C05472=1136.508,344.790,-80.424,-177.368,10.885,149.505
C05473=1136.503,345.037,-80.459,-177.365,10.887,149.505
C05474=1136.500,345.285,-80.494,-177.361,10.890,149.505
C05475=1136.495,345.532,-80.529,-177.358,10.892,149.504
C05476=1136.492,345.780,-80.563,-177.355,10.895,149.504
C05477=1136.488,346.027,-80.598,-177.351,10.897,149.504
C05478=1136.484,346.275,-80.633,-177.348,10.899,149.504
C05479=1136.480,346.523,-80.668,-177.345,10.902,149.503
C05480=1136.476,346.770,-80.702,-177.342,10.905,149.503
C05481=1136.472,347.018,-80.737,-177.338,10.907,149.503
C05482=1136.468,347.265,-80.772,-177.335,10.910,149.503
C05483=1136.464,347.513,-80.807,-177.332,10.912,149.503
C05484=1136.460,347.761,-80.842,-177.328,10.915,149.503
C05485=1136.458,347.974,-80.872,-177.325,10.917,149.502
C05486=1136.454,348.186,-80.902,-177.323,10.919,149.502
C05487=1136.450,348.400,-80.932,-177.320,10.921,149.502
C05488=1136.447,348.614,-80.963,-177.317,10.923,149.502
C05489=1136.443,348.827,-80.993,-177.314,10.926,149.502
C05490=1136.440,349.040,-81.022,-177.311,10.928,149.501
C05491=1136.437,349.254,-81.053,-177.309,10.930,149.501
C05492=1136.433,349.466,-81.083,-177.306,10.932,149.501
C05493=1136.429,349.714,-81.118,-177.302,10.935,149.501
C05494=1136.425,349.962,-81.154,-177.298,10.937,149.501
C05495=1136.421,350.209,-81.189,-177.294,10.941,149.500
C05496=1136.417,350.457,-81.224,-177.291,10.943,149.500
C05497=1136.413,350.704,-81.259,-177.286,10.946,149.500
C05498=1136.410,350.951,-81.293,-177.283,10.949,149.499
C05499=1136.406,351.199,-81.329,-177.279,10.952,149.499
C05500=1136.402,351.446,-81.364,-177.275,10.954,149.499
C05501=1136.399,351.694,-81.400,-177.272,10.957,149.499
C05502=1136.394,351.941,-81.434,-177.268,10.960,149.498
C05503=1136.390,352.189,-81.470,-177.264,10.962,149.498
C05504=1136.387,352.436,-81.505,-177.261,10.965,149.498
C05505=1136.383,352.684,-81.541,-177.257,10.967,149.498
C05506=1136.378,352.931,-81.575,-177.253,10.970,149.497
C05507=1136.375,353.179,-81.611,-177.250,10.973,149.497
C05508=1136.371,353.426,-81.646,-177.245,10.976,149.497
C05509=1136.368,353.674,-81.682,-177.242,10.978,149.496
C05510=1136.363,353.921,-81.717,-177.239,10.981,149.496
C05511=1136.359,354.169,-81.752,-177.234,10.984,149.496
C05512=1136.355,354.416,-81.788,-177.231,10.986,149.496
C05513=1136.351,354.664,-81.824,-177.228,10.988,149.495
C05514=1136.347,354.911,-81.859,-177.223,10.991,149.495
C05515=1136.343,355.158,-81.894,-177.220,10.994,149.495
C05516=1136.340,355.406,-81.930,-177.217,10.996,149.495
C05517=1136.336,355.653,-81.965,-177.213,10.998,149.494
C05518=1136.332,355.901,-82.001,-177.209,11.002,149.494
C05519=1136.329,356.148,-82.036,-177.206,11.004,149.494
C05520=1136.324,356.395,-82.072,-177.202,11.006,149.493
C05521=1136.320,356.643,-82.108,-177.199,11.009,149.493
C05522=1136.316,356.890,-82.143,-177.195,11.012,149.493
C05523=1136.313,357.138,-82.179,-177.191,11.014,149.493
C05524=1136.309,357.385,-82.214,-177.188,11.017,149.492
C05525=1136.305,357.633,-82.250,-177.184,11.019,149.492
C05526=1136.301,357.881,-82.286,-177.181,11.022,149.492
C05527=1136.297,358.127,-82.321,-177.177,11.024,149.492
C05528=1136.293,358.374,-82.358,-177.174,11.027,149.491
C05529=1136.290,358.622,-82.393,-177.170,11.029,149.491
C05530=1136.285,358.870,-82.429,-177.167,11.032,149.491
C05531=1136.282,359.117,-82.465,-177.163,11.034,149.490
C05532=1136.278,359.365,-82.500,-177.160,11.036,149.490
C05533=1136.275,359.612,-82.537,-177.157,11.039,149.490
C05534=1136.270,359.859,-82.573,-177.153,11.041,149.490
C05535=1136.266,360.107,-82.608,-177.150,11.044,149.489
C05536=1136.263,360.354,-82.644,-177.146,11.046,149.489
C05537=1136.259,360.601,-82.680,-177.143,11.048,149.489
C05538=1136.254,360.848,-82.716,-177.139,11.051,149.489
C05539=1136.251,361.096,-82.751,-177.135,11.054,149.488
C05540=1136.247,361.343,-82.787,-177.132,11.056,149.488
C05541=1136.243,361.556,-82.819,-177.129,11.058,149.488
C05542=1136.241,361.770,-82.850,-177.127,11.060,149.488
C05543=1136.238,361.983,-82.881,-177.123,11.062,149.487
C05544=1136.234,362.196,-82.912,-177.121,11.064,149.487
C05545=1136.231,362.409,-82.943,-177.117,11.066,149.487
C05546=1136.228,362.622,-82.973,-177.115,11.068,149.487
C05547=1136.224,362.835,-83.005,-177.111,11.070,149.486
C05548=1136.221,363.048,-83.036,-177.109,11.072,149.486
C05549=1136.217,363.295,-83.072,-177.105,11.075,149.486
C05550=1136.213,363.543,-83.108,-177.102,11.077,149.486
C05551=1136.210,363.790,-83.145,-177.099,11.080,149.486
C05552=1136.205,364.038,-83.181,-177.096,11.082,149.485
C05553=1136.202,364.285,-83.217,-177.092,11.085,149.485
C05554=1136.198,364.532,-83.253,-177.090,11.086,149.485
C05555=1136.194,364.779,-83.289,-177.086,11.088,149.484
C05556=1136.190,365.027,-83.325,-177.083,11.091,149.484
C05557=1136.186,365.274,-83.362,-177.079,11.093,149.484
C05558=1136.183,365.522,-83.397,-177.076,11.096,149.484
C05559=1136.179,365.769,-83.434,-177.073,11.098,149.484
C05560=1136.175,366.016,-83.470,-177.069,11.101,149.483
C05561=1136.171,366.263,-83.507,-177.067,11.102,149.483
C05562=1136.168,366.511,-83.543,-177.063,11.105,149.483
C05563=1136.164,366.759,-83.579,-177.060,11.107,149.483
C05564=1136.160,367.006,-83.616,-177.057,11.110,149.483
C05565=1136.156,367.253,-83.653,-177.053,11.112,149.482
C05566=1136.153,367.500,-83.688,-177.051,11.114,149.482
C05567=1136.148,367.748,-83.725,-177.047,11.116,149.482
C05568=1136.144,367.995,-83.762,-177.044,11.119,149.482
C05569=1136.141,368.242,-83.797,-177.041,11.121,149.481
C05570=1136.137,368.490,-83.834,-177.038,11.123,149.481
C05571=1136.133,368.736,-83.870,-177.035,11.126,149.481
C05572=1136.129,368.984,-83.907,-177.032,11.128,149.481
C05573=1136.125,369.232,-83.944,-177.029,11.130,149.481
C05574=1136.122,369.479,-83.980,-177.026,11.132,149.480
C05575=1136.118,369.726,-84.017,-177.022,11.135,149.480
C05576=1136.115,369.973,-84.053,-177.020,11.136,149.480
C05577=1136.110,370.220,-84.090,-177.016,11.139,149.480
C05578=1136.106,370.468,-84.126,-177.013,11.141,149.479
C05579=1136.103,370.715,-84.162,-177.010,11.143,149.479
C05580=1136.099,370.962,-84.199,-177.007,11.146,149.479
C05581=1136.095,371.210,-84.237,-177.004,11.148,149.479
C05582=1136.092,371.457,-84.273,-177.001,11.150,149.479
C05583=1136.088,371.704,-84.310,-176.998,11.152,149.479
C05584=1136.084,371.951,-84.347,-176.995,11.155,149.478
C05585=1136.079,372.198,-84.383,-176.992,11.157,149.478
C05586=1136.076,372.445,-84.420,-176.989,11.159,149.478
C05587=1136.073,372.693,-84.457,-176.987,11.161,149.478
C05588=1136.068,372.940,-84.494,-176.983,11.164,149.478
C05589=1136.065,373.187,-84.530,-176.980,11.166,149.477
C05590=1136.061,373.434,-84.567,-176.978,11.168,149.477
C05591=1136.057,373.682,-84.604,-176.974,11.171,149.477
C05592=1136.053,373.930,-84.641,-176.972,11.172,149.477
C05593=1136.049,374.177,-84.678,-176.969,11.175,149.477
C05594=1136.046,374.424,-84.714,-176.966,11.177,149.477
C05595=1136.042,374.671,-84.751,-176.963,11.179,149.476
C05596=1136.038,374.919,-84.788,-176.961,11.181,149.476
C05597=1136.035,375.131,-84.819,-176.958,11.183,149.476
C05598=1136.032,375.344,-84.851,-176.956,11.185,149.476
C05599=1136.028,375.557,-84.883,-176.953,11.187,149.476
C05600=1136.025,375.771,-84.915,-176.951,11.189,149.476
C05601=1136.022,375.983,-84.947,-176.948,11.191,149.476
C05602=1136.019,376.196,-84.979,-176.946,11.193,149.476
C05603=1136.016,376.409,-85.011,-176.944,11.195,149.475
C05604=1136.012,376.622,-85.043,-176.941,11.197,149.475
C05605=1136.008,376.869,-85.079,-176.938,11.199,149.475
C05606=1136.004,377.116,-85.116,-176.936,11.201,149.475
C05607=1136.001,377.364,-85.154,-176.933,11.204,149.475
C05608=1135.997,377.611,-85.191,-176.930,11.206,149.475
C05609=1135.993,377.858,-85.228,-176.927,11.208,149.475
C05610=1135.990,378.106,-85.265,-176.925,11.210,149.475
C05611=1135.986,378.353,-85.302,-176.922,11.212,149.474
C05612=1135.982,378.600,-85.339,-176.919,11.215,149.474
C05613=1135.978,378.847,-85.376,-176.917,11.217,149.474
C05614=1135.974,379.095,-85.413,-176.914,11.219,149.474
C05615=1135.971,379.341,-85.450,-176.912,11.221,149.474
C05616=1135.967,379.588,-85.487,-176.909,11.223,149.474
C05617=1135.963,379.836,-85.524,-176.906,11.226,149.474
C05618=1135.960,380.083,-85.562,-176.904,11.228,149.474
C05619=1135.956,380.330,-85.599,-176.901,11.230,149.474
C05620=1135.952,380.578,-85.636,-176.899,11.233,149.474
C05621=1135.948,380.824,-85.674,-176.896,11.235,149.473
C05622=1135.944,381.072,-85.710,-176.894,11.237,149.473
C05623=1135.941,381.319,-85.748,-176.891,11.239,149.473
C05624=1135.937,381.566,-85.785,-176.888,11.241,149.473
C05625=1135.933,381.813,-85.822,-176.886,11.243,149.473
C05626=1135.930,382.060,-85.860,-176.883,11.246,149.473
C05627=1135.925,382.308,-85.897,-176.881,11.248,149.473
C05628=1135.922,382.554,-85.934,-176.879,11.250,149.473
C05629=1135.918,382.802,-85.972,-176.876,11.253,149.473
C05630=1135.914,383.049,-86.009,-176.874,11.255,149.473
C05631=1135.911,383.297,-86.046,-176.871,11.257,149.473
C05632=1135.907,383.543,-86.084,-176.869,11.260,149.473
C05633=1135.902,383.791,-86.122,-176.869,11.260,149.473
C05634=1135.899,384.038,-86.159,-176.868,11.262,149.473
C05635=1135.895,384.285,-86.196,-176.867,11.264,149.474
C05636=1135.891,384.532,-86.234,-176.866,11.265,149.474
C05637=1135.888,384.780,-86.271,-176.865,11.266,149.474
C05638=1135.884,385.026,-86.309,-176.864,11.268,149.474
C05639=1135.881,385.273,-86.347,-176.863,11.269,149.474
C05640=1135.877,385.521,-86.383,-176.862,11.271,149.474
C05641=1135.873,385.767,-86.421,-176.862,11.273,149.475
C05642=1135.869,386.015,-86.458,-176.861,11.273,149.475
C05643=1135.866,386.262,-86.496,-176.860,11.275,149.475
C05644=1135.862,386.510,-86.533,-176.859,11.277,149.475
C05645=1135.858,386.756,-86.571,-176.858,11.279,149.475
C05646=1135.854,387.004,-86.609,-176.858,11.280,149.476
C05647=1135.850,387.251,-86.646,-176.857,11.282,149.476
C05648=1135.847,387.497,-86.684,-176.856,11.284,149.476
C05649=1135.843,387.745,-86.721,-176.856,11.285,149.476
C05650=1135.839,387.992,-86.758,-176.855,11.287,149.477
C05651=1135.836,388.239,-86.796,-176.854,11.289,149.477
C05652=1135.832,388.486,-86.833,-176.854,11.290,149.477
C05653=1135.828,388.699,-86.866,-176.853,11.292,149.478
C05654=1135.825,388.912,-86.898,-176.853,11.293,149.478
C05655=1135.822,389.125,-86.931,-176.852,11.295,149.478
C05656=1135.820,389.337,-86.963,-176.852,11.296,149.478
C05657=1135.816,389.550,-86.995,-176.852,11.297,149.478
C05658=1135.813,389.763,-87.028,-176.851,11.299,149.479
C05659=1135.809,389.976,-87.060,-176.851,11.300,149.479
C05660=1135.806,390.189,-87.092,-176.850,11.302,149.479
C05661=1135.803,390.436,-87.130,-176.850,11.304,149.480
C05662=1135.798,390.683,-87.167,-176.850,11.306,149.480
C05663=1135.795,390.931,-87.205,-176.849,11.308,149.480
C05664=1135.791,391.177,-87.243,-176.849,11.309,149.481
C05665=1135.788,391.425,-87.280,-176.849,11.311,149.481
C05666=1135.784,391.672,-87.317,-176.848,11.314,149.482
C05667=1135.780,391.919,-87.356,-176.848,11.315,149.482
C05668=1135.776,392.166,-87.393,-176.847,11.317,149.482
C05669=1135.773,392.414,-87.431,-176.847,11.319,149.483
C05670=1135.769,392.660,-87.468,-176.847,11.321,149.483
C05671=1135.765,392.907,-87.505,-176.847,11.323,149.484
C05672=1135.762,393.155,-87.543,-176.847,11.325,149.484
C05673=1135.757,393.402,-87.581,-176.847,11.327,149.485
C05674=1135.754,393.649,-87.619,-176.846,11.329,149.485
C05675=1135.750,393.896,-87.656,-176.846,11.331,149.486
C05676=1135.747,394.143,-87.694,-176.846,11.333,149.486
C05677=1135.743,394.390,-87.732,-176.846,11.335,149.487
C05678=1135.739,394.638,-87.769,-176.845,11.338,149.487
C05679=1135.735,394.885,-87.807,-176.846,11.339,149.488
C05680=1135.732,395.132,-87.845,-176.846,11.342,149.488
C05681=1135.728,395.378,-87.882,-176.845,11.344,149.489
C05682=1135.724,395.626,-87.919,-176.846,11.346,149.490
C05683=1135.720,395.873,-87.958,-176.846,11.348,149.490
C05684=1135.716,396.120,-87.995,-176.845,11.351,149.491
C05685=1135.713,396.367,-88.033,-176.845,11.353,149.491
C05686=1135.709,396.614,-88.070,-176.846,11.355,149.492
C05687=1135.706,396.862,-88.108,-176.846,11.358,149.493
C05688=1135.701,397.108,-88.146,-176.846,11.360,149.493
C05689=1135.698,397.356,-88.184,-176.846,11.362,149.494
C05690=1135.694,397.603,-88.221,-176.846,11.364,149.495
C05691=1135.691,397.850,-88.259,-176.846,11.367,149.495
C05692=1135.687,398.097,-88.297,-176.847,11.369,149.496
C05693=1135.683,398.344,-88.335,-176.847,11.371,149.496
C05694=1135.679,398.591,-88.373,-176.847,11.374,149.497
C05695=1135.676,398.839,-88.410,-176.847,11.377,149.498
C05696=1135.672,399.085,-88.448,-176.848,11.379,149.499
C05697=1135.668,399.333,-88.486,-176.848,11.381,149.499
C05698=1135.664,399.579,-88.524,-176.848,11.384,149.500
C05699=1135.661,399.827,-88.562,-176.848,11.387,149.501
C05700=1135.657,400.074,-88.598,-176.849,11.389,149.502
C05701=1135.653,400.321,-88.637,-176.849,11.392,149.502
C05702=1135.649,400.568,-88.675,-176.850,11.395,149.503
C05703=1135.646,400.815,-88.712,-176.851,11.397,149.504
C05704=1135.642,401.062,-88.750,-176.851,11.400,149.505
C05705=1135.638,401.309,-88.787,-176.851,11.403,149.506
C05706=1135.634,401.557,-88.825,-176.852,11.406,149.507
C05707=1135.631,401.803,-88.863,-176.853,11.408,149.507
C05708=1135.627,402.051,-88.901,-176.853,11.411,149.508
C05709=1135.624,402.263,-88.934,-176.853,11.413,149.509
C05710=1135.621,402.476,-88.967,-176.854,11.416,149.510
C05711=1135.617,402.689,-88.998,-176.854,11.418,149.510
C05712=1135.614,402.902,-89.031,-176.855,11.420,149.511
C05713=1135.611,403.114,-89.064,-176.855,11.423,149.512
C05714=1135.608,403.327,-89.097,-176.856,11.425,149.513
C05715=1135.605,403.540,-89.129,-176.857,11.428,149.514
C05716=1135.601,403.753,-89.162,-176.858,11.430,149.514
C05717=1135.598,404.000,-89.199,-176.858,11.433,149.515
C05718=1135.594,404.247,-89.237,-176.859,11.436,149.516
C05719=1135.591,404.494,-89.275,-176.859,11.439,149.517
C05720=1135.587,404.741,-89.313,-176.860,11.443,149.518
C05721=1135.583,404.988,-89.351,-176.861,11.445,149.519
C05722=1135.580,405.235,-89.389,-176.862,11.448,149.520
C05723=1135.576,405.482,-89.426,-176.863,11.452,149.521
C05724=1135.572,405.730,-89.464,-176.864,11.455,149.522
C05725=1135.568,405.977,-89.502,-176.865,11.458,149.523
C05726=1135.565,406.224,-89.540,-176.865,11.462,149.525
C05727=1135.560,406.471,-89.578,-176.867,11.464,149.525
C05728=1135.557,406.718,-89.616,-176.868,11.468,149.527
C05729=1135.553,406.965,-89.653,-176.868,11.471,149.528
C05730=1135.550,407.212,-89.691,-176.869,11.474,149.529
C05731=1135.546,407.459,-89.730,-176.871,11.478,149.530
C05732=1135.542,407.707,-89.767,-176.872,11.481,149.531
C05733=1135.538,407.953,-89.804,-176.872,11.485,149.532
C05734=1135.534,408.201,-89.843,-176.874,11.487,149.533
C05735=1135.531,408.447,-89.880,-176.875,11.491,149.535
C05736=1135.527,408.695,-89.918,-176.876,11.494,149.536
C05737=1135.524,408.942,-89.956,-176.877,11.498,149.537
C05738=1135.520,409.189,-89.995,-176.878,11.502,149.538
C05739=1135.516,409.436,-90.032,-176.880,11.505,149.540
C05740=1135.513,409.683,-90.070,-176.881,11.509,149.541
C05741=1135.509,409.930,-90.109,-176.882,11.513,149.542
C05742=1135.505,410.177,-90.146,-176.884,11.516,149.543
C05743=1135.502,410.424,-90.184,-176.885,11.520,149.545
C05744=1135.497,410.671,-90.222,-176.887,11.523,149.546
C05745=1135.494,410.919,-90.259,-176.888,11.527,149.547
C05746=1135.490,411.165,-90.297,-176.889,11.530,149.549
C05747=1135.487,411.413,-90.335,-176.891,11.534,149.550
C05748=1135.482,411.659,-90.373,-176.892,11.538,149.551
C05749=1135.479,411.907,-90.411,-176.894,11.542,149.553
C05750=1135.475,412.153,-90.449,-176.895,11.546,149.554
C05751=1135.471,412.401,-90.487,-176.897,11.550,149.555
C05752=1135.468,412.648,-90.525,-176.898,11.554,149.557
C05753=1135.464,412.895,-90.563,-176.900,11.558,149.558
C05754=1135.460,413.142,-90.601,-176.902,11.562,149.560
C05755=1135.457,413.389,-90.639,-176.903,11.566,149.561
C05756=1135.453,413.636,-90.677,-176.905,11.570,149.563
C05757=1135.449,413.883,-90.715,-176.907,11.574,149.564
C05758=1135.446,414.130,-90.753,-176.908,11.578,149.566
C05759=1135.442,414.377,-90.790,-176.910,11.582,149.567
C05760=1135.439,414.624,-90.828,-176.912,11.586,149.569
C05761=1135.437,414.872,-90.866,-176.914,11.591,149.570
C05762=1135.434,415.119,-90.903,-176.916,11.595,149.572
C05763=1135.434,415.365,-90.941,-176.918,11.599,149.573
C05764=1135.433,415.614,-90.979,-176.919,11.603,149.575
C05765=1135.433,415.826,-91.011,-176.921,11.607,149.576
C05766=1135.434,416.039,-91.044,-176.922,11.611,149.578
C05767=1135.435,416.251,-91.075,-176.925,11.615,149.579
C05768=1135.436,416.464,-91.107,-176.926,11.618,149.581
C05769=1135.439,416.677,-91.139,-176.928,11.622,149.582
C05770=1135.441,416.889,-91.171,-176.930,11.626,149.584
C05771=1135.444,417.102,-91.203,-176.932,11.630,149.585
C05772=1135.448,417.314,-91.234,-176.934,11.634,149.586
C05773=1135.029,417.314,-91.297,-176.926,11.638,149.586
C05774=1135.025,417.102,-91.266,-176.924,11.634,149.584
C05775=1135.022,416.889,-91.234,-176.922,11.631,149.583
C05776=1135.019,416.676,-91.202,-176.920,11.627,149.581
C05777=1135.018,416.463,-91.170,-176.919,11.623,149.580
C05778=1135.016,416.251,-91.138,-176.917,11.619,149.578
C05779=1135.015,416.038,-91.106,-176.915,11.616,149.577
C05780=1135.014,415.826,-91.074,-176.914,11.612,149.576
C05781=1135.014,415.614,-91.041,-176.912,11.608,149.574
C05782=1135.015,415.365,-91.004,-176.910,11.603,149.573
C05783=1135.016,415.119,-90.966,-176.908,11.599,149.571
C05784=1135.017,414.871,-90.928,-176.906,11.595,149.570
C05785=1135.020,414.624,-90.891,-176.905,11.591,149.568
C05786=1135.023,414.377,-90.852,-176.903,11.587,149.567
C05787=1135.026,414.130,-90.815,-176.901,11.583,149.565
C05788=1135.030,413.884,-90.777,-176.900,11.578,149.563
C05789=1135.034,413.636,-90.738,-176.899,11.574,149.562
C05790=1135.037,413.389,-90.701,-176.897,11.570,149.560
C05791=1135.041,413.142,-90.663,-176.895,11.566,149.559
C05792=1135.044,412.895,-90.624,-176.894,11.562,149.558
C05793=1135.048,412.648,-90.587,-176.892,11.558,149.556
C05794=1135.052,412.400,-90.550,-176.890,11.554,149.555
C05795=1135.056,412.153,-90.511,-176.889,11.550,149.553
C05796=1135.059,411.906,-90.473,-176.887,11.546,149.552
C05797=1135.063,411.659,-90.436,-176.886,11.542,149.551
C05798=1135.067,411.412,-90.397,-176.885,11.538,149.549
C05799=1135.071,411.165,-90.360,-176.883,11.535,149.548
C05800=1135.074,410.918,-90.322,-176.882,11.531,149.547
C05801=1135.079,410.671,-90.284,-176.880,11.527,149.545
C05802=1135.082,410.424,-90.246,-176.879,11.523,149.544
C05803=1135.085,410.177,-90.208,-176.878,11.519,149.543
C05804=1135.090,409.930,-90.170,-176.877,11.516,149.542
C05805=1135.093,409.682,-90.132,-176.876,11.512,149.540
C05806=1135.097,409.436,-90.094,-176.874,11.508,149.539
C05807=1135.101,409.188,-90.056,-176.873,11.505,149.538
C05808=1135.104,408.942,-90.018,-176.872,11.501,149.537
C05809=1135.107,408.694,-89.980,-176.871,11.498,149.535
C05810=1135.111,408.448,-89.942,-176.870,11.494,149.534
C05811=1135.115,408.200,-89.904,-176.869,11.491,149.533
C05812=1135.119,407.954,-89.866,-176.868,11.487,149.532
C05813=1135.122,407.706,-89.828,-176.867,11.484,149.531
C05814=1135.127,407.459,-89.791,-176.866,11.480,149.530
C05815=1135.130,407.212,-89.753,-176.864,11.478,149.528
C05816=1135.133,406.964,-89.715,-176.863,11.474,149.527
C05817=1135.138,406.718,-89.677,-176.862,11.471,149.526
C05818=1135.141,406.470,-89.639,-176.862,11.468,149.525
C05819=1135.145,406.224,-89.601,-176.861,11.464,149.524
C05820=1135.148,405.976,-89.563,-176.860,11.461,149.523
C05821=1135.153,405.730,-89.525,-176.859,11.458,149.522
C05822=1135.156,405.482,-89.487,-176.858,11.454,149.521
C05823=1135.160,405.236,-89.450,-176.857,11.451,149.520
C05824=1135.163,404.988,-89.411,-176.856,11.448,149.519
C05825=1135.168,404.741,-89.374,-176.856,11.446,149.518
C05826=1135.171,404.494,-89.336,-176.855,11.442,149.517
C05827=1135.175,404.247,-89.299,-176.854,11.439,149.516
C05828=1135.178,403.999,-89.260,-176.854,11.436,149.515
C05829=1135.182,403.753,-89.223,-176.853,11.433,149.514
C05830=1135.185,403.540,-89.190,-176.852,11.431,149.513
C05831=1135.189,403.328,-89.157,-176.852,11.428,149.512
C05832=1135.192,403.114,-89.124,-176.851,11.426,149.512
C05833=1135.195,402.902,-89.092,-176.851,11.423,149.511
C05834=1135.197,402.689,-89.060,-176.850,11.420,149.510
C05835=1135.201,402.476,-89.027,-176.849,11.418,149.509
C05836=1135.204,402.264,-88.995,-176.850,11.416,149.509
C05837=1135.207,402.051,-88.962,-176.849,11.413,149.508
C05838=1135.211,401.804,-88.925,-176.848,11.411,149.507
C05839=1135.215,401.556,-88.887,-176.848,11.408,149.506
C05840=1135.219,401.310,-88.849,-176.848,11.405,149.505
C05841=1135.222,401.062,-88.811,-176.847,11.402,149.504
C05842=1135.226,400.816,-88.773,-176.846,11.400,149.504
C05843=1135.230,400.568,-88.735,-176.846,11.397,149.503
C05844=1135.234,400.321,-88.698,-176.846,11.394,149.502
C05845=1135.237,400.074,-88.660,-176.845,11.391,149.501
C05846=1135.241,399.827,-88.623,-176.845,11.389,149.501
C05847=1135.245,399.580,-88.584,-176.844,11.386,149.500
C05848=1135.249,399.333,-88.546,-176.844,11.384,149.499
C05849=1135.252,399.086,-88.508,-176.844,11.381,149.498
C05850=1135.256,398.839,-88.472,-176.844,11.378,149.498
C05851=1135.260,398.591,-88.433,-176.843,11.376,149.497
C05852=1135.264,398.344,-88.396,-176.843,11.374,149.496
C05853=1135.267,398.097,-88.358,-176.843,11.371,149.496
C05854=1135.271,397.851,-88.320,-176.843,11.368,149.495
C05855=1135.275,397.602,-88.282,-176.843,11.367,149.494
C05856=1135.279,397.356,-88.245,-176.843,11.364,149.493
C05857=1135.282,397.109,-88.207,-176.843,11.361,149.493
C05858=1135.286,396.862,-88.169,-176.843,11.359,149.492
C05859=1135.289,396.615,-88.131,-176.842,11.357,149.492
C05860=1135.294,396.367,-88.094,-176.842,11.355,149.491
C05861=1135.297,396.120,-88.056,-176.843,11.352,149.490
C05862=1135.301,395.873,-88.018,-176.843,11.350,149.490
C05863=1135.304,395.626,-87.980,-176.842,11.348,149.489
C05864=1135.309,395.379,-87.943,-176.843,11.346,149.489
C05865=1135.313,395.132,-87.905,-176.843,11.343,149.488
C05866=1135.316,394.885,-87.867,-176.843,11.341,149.488
C05867=1135.320,394.638,-87.830,-176.843,11.339,149.487
C05868=1135.323,394.390,-87.792,-176.843,11.337,149.487
C05869=1135.328,394.143,-87.754,-176.843,11.334,149.486
C05870=1135.331,393.896,-87.716,-176.843,11.333,149.486
C05871=1135.334,393.650,-87.679,-176.844,11.331,149.485
C05872=1135.338,393.402,-87.642,-176.844,11.329,149.485
C05873=1135.342,393.155,-87.604,-176.844,11.326,149.484
C05874=1135.345,392.908,-87.566,-176.844,11.325,149.484
C05875=1135.350,392.660,-87.529,-176.844,11.322,149.483
C05876=1135.353,392.413,-87.491,-176.845,11.320,149.483
C05877=1135.357,392.167,-87.453,-176.845,11.319,149.482
C05878=1135.361,391.919,-87.416,-176.846,11.317,149.482
C05879=1135.364,391.672,-87.378,-176.846,11.315,149.481
C05880=1135.368,391.426,-87.341,-176.846,11.312,149.481
C05881=1135.372,391.178,-87.302,-176.846,11.311,149.481
C05882=1135.376,390.931,-87.265,-176.847,11.309,149.480
C05883=1135.379,390.683,-87.227,-176.848,11.307,149.480
C05884=1135.383,390.437,-87.190,-176.848,11.306,149.480
C05885=1135.386,390.189,-87.153,-176.848,11.303,149.479
C05886=1135.390,389.977,-87.120,-176.849,11.301,149.479
C05887=1135.394,389.764,-87.088,-176.849,11.300,149.479
C05888=1135.396,389.551,-87.055,-176.850,11.298,149.478
C05889=1135.399,389.339,-87.023,-176.850,11.297,149.478
C05890=1135.402,389.125,-86.991,-176.850,11.296,149.478
C05891=1135.406,388.913,-86.958,-176.851,11.294,149.477
C05892=1135.409,388.699,-86.926,-176.851,11.293,149.477
C05893=1135.413,388.487,-86.894,-176.852,11.291,149.477
C05894=1135.416,388.240,-86.856,-176.853,11.289,149.477
C05895=1135.420,387.992,-86.819,-176.853,11.288,149.476
C05896=1135.424,387.746,-86.781,-176.854,11.286,149.476
C05897=1135.427,387.498,-86.743,-176.855,11.284,149.476
C05898=1135.431,387.251,-86.706,-176.855,11.283,149.476
C05899=1135.435,387.005,-86.669,-176.856,11.281,149.475
C05900=1135.438,386.757,-86.632,-176.857,11.279,149.475
C05901=1135.442,386.510,-86.594,-176.858,11.278,149.475
C05902=1135.445,386.263,-86.556,-176.858,11.277,149.475
C05903=1135.450,386.015,-86.519,-176.859,11.275,149.475
C05904=1135.453,385.768,-86.481,-176.861,11.273,149.474
C05905=1135.457,385.521,-86.444,-176.861,11.272,149.474
C05906=1135.461,385.274,-86.406,-176.862,11.270,149.474
C05907=1135.465,385.026,-86.369,-176.863,11.268,149.474
C05908=1135.468,384.780,-86.331,-176.864,11.267,149.474
C05909=1135.472,384.532,-86.294,-176.864,11.266,149.474
C05910=1135.476,384.285,-86.257,-176.866,11.264,149.473
C05911=1135.479,384.039,-86.219,-176.866,11.262,149.473
C05912=1135.483,383.791,-86.182,-176.867,11.262,149.473
C05913=1135.487,383.544,-86.144,-176.868,11.260,149.473
C05914=1135.491,383.297,-86.107,-176.870,11.258,149.473
C05915=1135.494,383.050,-86.069,-176.873,11.256,149.473
C05916=1135.498,382.803,-86.033,-176.875,11.254,149.473
C05917=1135.501,382.555,-85.995,-176.877,11.252,149.473
C05918=1135.506,382.308,-85.957,-176.880,11.249,149.473
C05919=1135.510,382.061,-85.920,-176.882,11.247,149.473
C05920=1135.513,381.813,-85.882,-176.885,11.245,149.473
C05921=1135.517,381.566,-85.846,-176.887,11.242,149.473
C05922=1135.521,381.320,-85.808,-176.890,11.240,149.473
C05923=1135.525,381.072,-85.771,-176.892,11.238,149.474
C05924=1135.529,380.825,-85.733,-176.895,11.235,149.474
C05925=1135.533,380.578,-85.696,-176.898,11.233,149.474
C05926=1135.535,380.330,-85.660,-176.900,11.230,149.474
C05927=1135.539,380.084,-85.622,-176.903,11.228,149.474
C05928=1135.543,379.837,-85.585,-176.905,11.227,149.474
C05929=1135.547,379.589,-85.548,-176.908,11.224,149.474
C05930=1135.551,379.342,-85.510,-176.911,11.222,149.474
C05931=1135.555,379.095,-85.474,-176.913,11.219,149.474
C05932=1135.558,378.847,-85.436,-176.916,11.217,149.474
C05933=1135.562,378.601,-85.399,-176.918,11.215,149.474
C05934=1135.566,378.353,-85.362,-176.921,11.213,149.474
C05935=1135.570,378.105,-85.325,-176.924,11.211,149.475
C05936=1135.574,377.858,-85.288,-176.927,11.208,149.475
C05937=1135.577,377.612,-85.250,-176.930,11.206,149.475
C05938=1135.581,377.365,-85.213,-176.932,11.204,149.475
C05939=1135.585,377.117,-85.176,-176.935,11.202,149.475
C05940=1135.588,376.870,-85.140,-176.937,11.200,149.475
C05941=1135.592,376.623,-85.102,-176.941,11.197,149.475
C05942=1135.596,376.410,-85.071,-176.943,11.195,149.475
C05943=1135.598,376.197,-85.039,-176.945,11.193,149.475
C05944=1135.602,375.984,-85.007,-176.947,11.191,149.476
C05945=1135.606,375.771,-84.975,-176.950,11.190,149.476
C05946=1135.608,375.558,-84.943,-176.952,11.188,149.476
C05947=1135.612,375.345,-84.912,-176.955,11.185,149.476
C05948=1135.615,375.133,-84.880,-176.957,11.184,149.476
C05949=1135.619,374.920,-84.848,-176.960,11.182,149.476
C05950=1135.622,374.672,-84.811,-176.962,11.180,149.476
C05951=1135.626,374.425,-84.774,-176.965,11.177,149.476
C05952=1135.630,374.178,-84.737,-176.969,11.175,149.477
C05953=1135.634,373.930,-84.701,-176.971,11.173,149.477
C05954=1135.638,373.683,-84.664,-176.974,11.170,149.477
C05955=1135.641,373.436,-84.627,-176.977,11.169,149.477
C05956=1135.645,373.188,-84.590,-176.980,11.166,149.477
C05957=1135.649,372.941,-84.553,-176.983,11.164,149.478
C05958=1135.653,372.694,-84.516,-176.986,11.162,149.478
C05959=1135.656,372.447,-84.480,-176.989,11.159,149.478
C05960=1135.660,372.199,-84.443,-176.992,11.157,149.478
C05961=1135.664,371.952,-84.406,-176.995,11.155,149.478
C05962=1135.668,371.705,-84.369,-176.998,11.153,149.479
C05963=1135.671,371.458,-84.333,-177.000,11.150,149.479
C05964=1135.675,371.211,-84.296,-177.004,11.148,149.479
C05965=1135.679,370.963,-84.259,-177.006,11.146,149.479
C05966=1135.682,370.715,-84.223,-177.010,11.144,149.479
C05967=1135.687,370.468,-84.187,-177.013,11.141,149.479
C05968=1135.691,370.221,-84.150,-177.016,11.140,149.480
C05969=1135.694,369.974,-84.113,-177.019,11.137,149.480
C05970=1135.698,369.727,-84.077,-177.022,11.134,149.480
C05971=1135.702,369.480,-84.040,-177.025,11.133,149.480
C05972=1135.706,369.232,-84.004,-177.028,11.130,149.480
C05973=1135.709,368.984,-83.967,-177.031,11.128,149.481
C05974=1135.713,368.738,-83.931,-177.034,11.126,149.481
C05975=1135.717,368.490,-83.894,-177.037,11.124,149.481
C05976=1135.721,368.243,-83.858,-177.040,11.121,149.481
C05977=1135.725,367.996,-83.821,-177.044,11.119,149.481
C05978=1135.729,367.748,-83.785,-177.046,11.117,149.482
C05979=1135.732,367.502,-83.748,-177.050,11.114,149.482
C05980=1135.736,367.254,-83.712,-177.053,11.112,149.482
C05981=1135.740,367.007,-83.676,-177.056,11.109,149.482
C05982=1135.744,366.760,-83.639,-177.060,11.107,149.483
C05983=1135.748,366.512,-83.603,-177.062,11.105,149.483
C05984=1135.751,366.264,-83.566,-177.066,11.103,149.483
C05985=1135.755,366.016,-83.530,-177.069,11.101,149.483
C05986=1135.759,365.770,-83.494,-177.073,11.098,149.484
C05987=1135.763,365.522,-83.457,-177.076,11.096,149.484
C05988=1135.767,365.275,-83.421,-177.079,11.094,149.484
C05989=1135.770,365.028,-83.385,-177.082,11.092,149.484
C05990=1135.774,364.780,-83.349,-177.085,11.089,149.485
C05991=1135.778,364.533,-83.313,-177.089,11.087,149.485
C05992=1135.782,364.286,-83.277,-177.092,11.084,149.485
C05993=1135.785,364.039,-83.240,-177.095,11.082,149.485
C05994=1135.790,363.791,-83.204,-177.099,11.080,149.486
C05995=1135.793,363.544,-83.168,-177.102,11.077,149.486
C05996=1135.797,363.296,-83.132,-177.105,11.075,149.486
C05997=1135.801,363.049,-83.096,-177.109,11.072,149.486
C05998=1135.804,362.836,-83.065,-177.111,11.070,149.486
C05999=1135.807,362.623,-83.034,-177.114,11.069,149.487
C06000=1135.811,362.410,-83.003,-177.117,11.066,149.487
C06001=1135.814,362.197,-82.971,-177.120,11.065,149.487
C06002=1135.818,361.984,-82.941,-177.123,11.062,149.487
C06003=1135.821,361.771,-82.909,-177.126,11.060,149.488
C06004=1135.824,361.558,-82.879,-177.128,11.058,149.488
C06005=1135.827,361.344,-82.848,-177.132,11.056,149.488
C06006=1135.832,361.097,-82.811,-177.135,11.054,149.488
C06007=1135.835,360.850,-82.776,-177.139,11.051,149.489
C06008=1135.839,360.602,-82.740,-177.142,11.049,149.489
C06009=1135.843,360.355,-82.704,-177.145,11.046,149.489
C06010=1135.847,360.108,-82.668,-177.149,11.044,149.489
C06011=1135.850,359.860,-82.632,-177.152,11.042,149.490
C06012=1135.854,359.613,-82.597,-177.156,11.039,149.490
C06013=1135.858,359.366,-82.560,-177.159,11.037,149.490
C06014=1135.862,359.118,-82.524,-177.163,11.035,149.490
C06015=1135.866,358.871,-82.489,-177.167,11.032,149.491
C06016=1135.869,358.623,-82.453,-177.170,11.029,149.491
C06017=1135.874,358.375,-82.417,-177.174,11.027,149.491
C06018=1135.877,358.128,-82.382,-177.177,11.024,149.492
C06019=1135.881,357.882,-82.346,-177.180,11.022,149.492
C06020=1135.885,357.634,-82.310,-177.183,11.020,149.492
C06021=1135.889,357.387,-82.275,-177.187,11.017,149.492
C06022=1135.893,357.139,-82.239,-177.191,11.014,149.493
C06023=1135.897,356.891,-82.203,-177.194,11.012,149.493
C06024=1135.900,356.644,-82.167,-177.198,11.010,149.493
C06025=1135.904,356.396,-82.132,-177.201,11.007,149.493
C06026=1135.908,356.149,-82.097,-177.205,11.004,149.494
C06027=1135.912,355.902,-82.061,-177.209,11.002,149.494
C06028=1135.916,355.654,-82.025,-177.212,10.999,149.494
C06029=1135.920,355.407,-81.989,-177.216,10.997,149.494
C06030=1135.924,355.159,-81.954,-177.220,10.994,149.495
C06031=1135.928,354.912,-81.919,-177.223,10.991,149.495
C06032=1135.931,354.665,-81.883,-177.227,10.989,149.495
C06033=1135.935,354.417,-81.848,-177.230,10.987,149.496
C06034=1135.939,354.169,-81.813,-177.234,10.984,149.496
C06035=1135.943,353.922,-81.777,-177.238,10.981,149.496
C06036=1135.947,353.675,-81.742,-177.241,10.979,149.496
C06037=1135.951,353.427,-81.707,-177.245,10.976,149.497
C06038=1135.954,353.180,-81.671,-177.249,10.973,149.497
C06039=1135.958,352.932,-81.635,-177.253,10.970,149.497
C06040=1135.963,352.685,-81.601,-177.256,10.968,149.497
C06041=1135.966,352.437,-81.565,-177.260,10.965,149.498
C06042=1135.970,352.190,-81.530,-177.264,10.963,149.498
C06043=1135.974,351.942,-81.494,-177.267,10.960,149.498
C06044=1135.978,351.695,-81.460,-177.271,10.957,149.498
C06045=1135.982,351.448,-81.424,-177.275,10.955,149.499
C06046=1135.985,351.200,-81.389,-177.279,10.951,149.499
C06047=1135.990,350.953,-81.354,-177.282,10.949,149.499
C06048=1135.994,350.705,-81.319,-177.286,10.946,149.500
C06049=1135.997,350.458,-81.283,-177.290,10.944,149.500
C06050=1136.001,350.210,-81.248,-177.294,10.940,149.500
C06051=1136.006,349.963,-81.213,-177.297,10.938,149.501
C06052=1136.009,349.715,-81.178,-177.301,10.935,149.501
C06053=1136.013,349.467,-81.143,-177.305,10.933,149.501
C06054=1136.017,349.255,-81.113,-177.308,10.930,149.501
C06055=1136.020,349.042,-81.083,-177.311,10.928,149.501
C06056=1136.023,348.828,-81.053,-177.314,10.926,149.501
C06057=1136.027,348.614,-81.022,-177.316,10.924,149.502
C06058=1136.030,348.401,-80.992,-177.320,10.921,149.502
C06059=1136.033,348.187,-80.962,-177.322,10.919,149.502
C06060=1136.037,347.975,-80.932,-177.325,10.918,149.502
C06061=1136.040,347.762,-80.902,-177.327,10.915,149.502
C06062=1136.044,347.514,-80.867,-177.331,10.913,149.503
C06063=1136.049,347.267,-80.832,-177.334,10.910,149.503
C06064=1136.052,347.019,-80.797,-177.337,10.908,149.503
C06065=1136.056,346.771,-80.762,-177.341,10.905,149.503
C06066=1136.060,346.524,-80.727,-177.344,10.903,149.504
C06067=1136.064,346.276,-80.693,-177.347,10.900,149.504
C06068=1136.068,346.029,-80.657,-177.351,10.898,149.504
C06069=1136.072,345.781,-80.623,-177.354,10.895,149.504
C06070=1136.076,345.534,-80.589,-177.357,10.893,149.504
C06071=1136.080,345.286,-80.553,-177.360,10.890,149.504
C06072=1136.084,345.038,-80.518,-177.363,10.888,149.505
C06073=1136.088,344.791,-80.484,-177.367,10.885,149.505
C06074=1136.091,344.544,-80.449,-177.370,10.883,149.505
C06075=1136.096,344.296,-80.414,-177.373,10.880,149.505
C06076=1136.099,344.048,-80.380,-177.377,10.878,149.506
C06077=1136.104,343.801,-80.346,-177.380,10.875,149.506
C06078=1136.108,343.553,-80.311,-177.383,10.873,149.506
C06079=1136.111,343.306,-80.276,-177.386,10.870,149.506
C06080=1136.115,343.058,-80.241,-177.390,10.868,149.506
C06081=1136.120,342.811,-80.207,-177.393,10.865,149.507
C06082=1136.123,342.563,-80.173,-177.396,10.863,149.507
C06083=1136.127,342.316,-80.138,-177.400,10.860,149.507
C06084=1136.131,342.067,-80.103,-177.402,10.858,149.507
C06085=1136.135,341.821,-80.069,-177.406,10.855,149.507
C06086=1136.139,341.573,-80.034,-177.409,10.853,149.508
C06087=1136.144,341.325,-80.000,-177.412,10.850,149.508
C06088=1136.147,341.078,-79.965,-177.416,10.848,149.508
C06089=1136.151,340.830,-79.931,-177.419,10.845,149.508
C06090=1136.155,340.582,-79.897,-177.421,10.843,149.508
C06091=1136.159,340.335,-79.862,-177.425,10.841,149.509
C06092=1136.163,340.087,-79.827,-177.428,10.838,149.509
C06093=1136.167,339.840,-79.793,-177.431,10.836,149.509
C06094=1136.171,339.592,-79.759,-177.435,10.833,149.509
C06095=1136.175,339.345,-79.725,-177.438,10.831,149.509
C06096=1136.179,339.097,-79.690,-177.441,10.828,149.510
C06097=1136.183,338.849,-79.656,-177.444,10.826,149.510
C06098=1136.187,338.602,-79.622,-177.447,10.823,149.510
C06099=1136.190,338.354,-79.587,-177.451,10.821,149.510
C06100=1136.195,338.107,-79.553,-177.454,10.818,149.511
C06101=1136.199,337.859,-79.520,-177.457,10.816,149.511
C06102=1136.203,337.611,-79.485,-177.460,10.813,149.511
C06103=1136.207,337.364,-79.451,-177.464,10.811,149.511
C06104=1136.211,337.116,-79.416,-177.467,10.808,149.511
C06105=1136.215,336.868,-79.382,-177.470,10.806,149.512
C06106=1136.218,336.621,-79.348,-177.473,10.803,149.512
C06107=1136.223,336.373,-79.314,-177.477,10.801,149.512
C06108=1136.227,336.125,-79.280,-177.480,10.798,149.512
C06109=1136.231,335.877,-79.246,-177.483,10.796,149.512
C06110=1136.234,335.664,-79.217,-177.486,10.793,149.512
C06111=1136.237,335.451,-79.188,-177.489,10.791,149.513
C06112=1136.241,335.238,-79.158,-177.491,10.789,149.513
C06113=1136.244,335.024,-79.129,-177.494,10.787,149.513
C06114=1136.247,334.811,-79.100,-177.497,10.785,149.513
C06115=1136.251,334.597,-79.070,-177.500,10.782,149.513
C06116=1136.254,334.384,-79.041,-177.502,10.780,149.513
C06117=1136.258,334.171,-79.012,-177.506,10.778,149.514
C06118=1136.262,333.923,-78.977,-177.509,10.775,149.514
C06119=1136.266,333.675,-78.944,-177.512,10.773,149.514
C06120=1136.270,333.428,-78.910,-177.515,10.770,149.514
C06121=1136.274,333.180,-78.875,-177.519,10.768,149.514
C06122=1136.278,332.932,-78.842,-177.521,10.766,149.515
C06123=1136.282,332.685,-78.808,-177.525,10.764,149.515
C06124=1136.286,332.437,-78.775,-177.527,10.761,149.515
C06125=1136.290,332.189,-78.740,-177.531,10.758,149.515
C06126=1136.294,331.941,-78.707,-177.534,10.756,149.516
C06127=1136.298,331.694,-78.673,-177.537,10.754,149.516
C06128=1136.301,331.446,-78.640,-177.540,10.751,149.516
C06129=1136.306,331.198,-78.605,-177.544,10.748,149.516
C06130=1136.310,330.951,-78.572,-177.547,10.746,149.516
C06131=1136.314,330.704,-78.538,-177.550,10.743,149.517
C06132=1136.317,330.455,-78.505,-177.553,10.741,149.517
C06133=1136.322,330.208,-78.470,-177.557,10.738,149.517
C06134=1136.326,329.960,-78.437,-177.560,10.736,149.517
C06135=1136.330,329.713,-78.403,-177.563,10.733,149.517
C06136=1136.333,329.464,-78.370,-177.566,10.730,149.517
C06137=1136.338,329.217,-78.336,-177.569,10.728,149.518
C06138=1136.341,328.970,-78.303,-177.573,10.726,149.518
C06139=1136.346,328.722,-78.269,-177.576,10.723,149.518
C06140=1136.350,328.474,-78.236,-177.579,10.720,149.518
C06141=1136.354,328.226,-78.201,-177.582,10.718,149.518
C06142=1136.358,327.978,-78.168,-177.586,10.715,149.519
C06143=1136.362,327.731,-78.135,-177.589,10.713,149.519
C06144=1136.366,327.483,-78.101,-177.592,10.710,149.519
C06145=1136.370,327.236,-78.068,-177.595,10.708,149.519
C06146=1136.374,326.988,-78.035,-177.598,10.705,149.519
C06147=1136.378,326.740,-78.001,-177.601,10.703,149.520
C06148=1136.381,326.492,-77.968,-177.605,10.700,149.520
C06149=1136.386,326.245,-77.934,-177.608,10.698,149.520
C06150=1136.390,325.997,-77.901,-177.611,10.695,149.520
C06151=1136.395,325.749,-77.868,-177.614,10.692,149.520
C06152=1136.399,325.501,-77.834,-177.618,10.690,149.521
C06153=1136.402,325.253,-77.801,-177.621,10.687,149.521
C06154=1136.406,325.006,-77.767,-177.624,10.685,149.521
C06155=1136.410,324.758,-77.734,-177.627,10.682,149.521
C06156=1136.414,324.510,-77.701,-177.630,10.680,149.521
C06157=1136.418,324.262,-77.667,-177.633,10.677,149.522
C06158=1136.423,324.015,-77.634,-177.637,10.675,149.522
C06159=1136.426,323.767,-77.602,-177.640,10.672,149.522
C06160=1136.430,323.520,-77.569,-177.642,10.670,149.522
C06161=1136.434,323.272,-77.535,-177.646,10.668,149.522
C06162=1136.438,323.023,-77.502,-177.649,10.665,149.523
C06163=1136.442,322.776,-77.469,-177.652,10.663,149.523
C06164=1136.446,322.528,-77.436,-177.655,10.660,149.523
C06165=1136.450,322.280,-77.402,-177.659,10.658,149.523
C06166=1136.454,322.047,-77.371,-177.662,10.655,149.523
C06167=1136.458,321.814,-77.340,-177.665,10.653,149.523
C06168=1136.462,321.581,-77.309,-177.668,10.650,149.524
C06169=1136.465,321.349,-77.278,-177.671,10.648,149.524
C06170=1136.469,321.115,-77.247,-177.673,10.645,149.524
C06171=1136.473,320.882,-77.216,-177.677,10.643,149.524
C06172=1136.477,320.649,-77.185,-177.679,10.641,149.524
C06173=1136.480,320.416,-77.154,-177.682,10.638,149.525
C06174=1136.485,320.168,-77.120,-177.686,10.636,149.525
C06175=1136.488,319.921,-77.088,-177.689,10.633,149.525
C06176=1136.492,319.673,-77.055,-177.692,10.631,149.525
C06177=1136.497,319.425,-77.022,-177.695,10.628,149.525
C06178=1136.501,319.177,-76.989,-177.698,10.626,149.525
C06179=1136.505,318.929,-76.956,-177.702,10.623,149.526
C06180=1136.508,318.682,-76.923,-177.705,10.621,149.526
C06181=1136.513,318.434,-76.891,-177.708,10.618,149.526
C06182=1136.517,318.186,-76.858,-177.711,10.615,149.526
C06183=1136.521,317.938,-76.825,-177.714,10.613,149.526
C06184=1136.525,317.690,-76.793,-177.717,10.610,149.527
C06185=1136.529,317.442,-76.760,-177.721,10.608,149.527
C06186=1136.547,316.329,-76.611,-176.869,8.949,148.880
C06187=1136.550,316.107,-76.582,-176.872,8.946,148.880
C06188=1136.554,315.885,-76.554,-176.874,8.942,148.880
C06189=1136.558,315.663,-76.525,-176.876,8.939,148.880
C06190=1136.562,315.415,-76.492,-176.879,8.936,148.879
C06191=1136.566,315.167,-76.460,-176.882,8.932,148.879
C06192=1136.570,314.919,-76.427,-176.884,8.928,148.879
C06193=1136.574,314.672,-76.396,-176.887,8.924,148.879
C06194=1136.579,314.424,-76.363,-176.889,8.921,148.879
C06195=1136.583,314.176,-76.331,-176.892,8.917,148.878
C06196=1136.587,313.928,-76.298,-176.894,8.914,148.878
C06197=1136.590,313.680,-76.266,-176.897,8.910,148.878
C06198=1136.595,313.402,-76.230,-176.900,8.906,148.878
C06199=1136.600,313.124,-76.195,-176.903,8.902,148.878
C06200=1136.604,312.846,-76.158,-176.907,8.898,148.878
C06201=1136.610,312.567,-76.122,-176.910,8.894,148.877
C06202=1136.613,312.320,-76.090,-176.913,8.890,148.877
C06203=1136.617,312.073,-76.058,-176.915,8.886,148.877
C06204=1136.622,311.824,-76.026,-176.918,8.882,148.877
C06205=1136.625,311.576,-75.994,-176.920,8.879,148.877
C06206=1136.629,311.328,-75.962,-176.923,8.875,148.876
C06207=1136.634,311.081,-75.930,-176.925,8.872,148.876
C06208=1136.638,310.833,-75.898,-176.928,8.869,148.876
C06209=1136.642,310.584,-75.867,-176.931,8.864,148.876
C06210=1136.647,310.337,-75.834,-176.933,8.861,148.876
C06211=1136.650,310.089,-75.803,-176.936,8.857,148.875
C06212=1136.654,309.841,-75.771,-176.939,8.854,148.875
C06213=1136.659,309.592,-75.738,-176.942,8.850,148.875
C06214=1136.663,309.345,-75.707,-176.944,8.847,148.875
C06215=1136.667,309.097,-75.675,-176.947,8.843,148.875
C06216=1136.670,308.849,-75.643,-176.949,8.840,148.875
C06217=1136.675,308.601,-75.611,-176.952,8.836,148.874
C06218=1136.679,308.353,-75.579,-176.955,8.832,148.874
C06219=1136.684,308.105,-75.548,-176.958,8.828,148.874
C06220=1136.687,307.857,-75.517,-176.960,8.825,148.874
C06221=1136.692,307.609,-75.484,-176.963,8.821,148.874
C06222=1136.696,307.362,-75.453,-176.966,8.818,148.874
C06223=1136.700,307.114,-75.421,-176.968,8.815,148.873
C06224=1136.704,306.866,-75.389,-176.971,8.811,148.873
C06225=1136.708,306.618,-75.358,-176.973,8.807,148.873
C06226=1136.713,306.369,-75.326,-176.977,8.804,148.873
C06227=1136.717,306.122,-75.294,-176.979,8.800,148.873
C06228=1136.721,305.874,-75.262,-176.982,8.796,148.873
C06229=1136.725,305.625,-75.231,-176.984,8.793,148.872
C06230=1136.729,305.378,-75.200,-176.987,8.789,148.872
C06231=1136.733,305.130,-75.168,-176.990,8.786,148.872
C06232=1136.738,304.882,-75.137,-176.992,8.783,148.872
C06233=1136.742,304.634,-75.105,-176.995,8.779,148.872
C06234=1136.746,304.386,-75.073,-176.998,8.775,148.872
C06235=1136.750,304.138,-75.042,-177.001,8.771,148.871
C06236=1136.754,303.889,-75.010,-177.003,8.768,148.871
C06237=1136.758,303.642,-74.979,-177.006,8.764,148.871
C06238=1136.762,303.393,-74.948,-177.009,8.761,148.871
C06239=1136.766,303.146,-74.916,-177.011,8.758,148.871
C06240=1136.770,302.897,-74.885,-177.014,8.754,148.871
C06241=1136.775,302.650,-74.854,-177.016,8.751,148.871
C06242=1136.779,302.401,-74.823,-177.020,8.747,148.871
C06243=1136.783,302.154,-74.791,-177.022,8.744,148.870
C06244=1136.787,301.905,-74.760,-177.025,8.740,148.870
C06245=1136.791,301.658,-74.728,-177.027,8.736,148.870
C06246=1136.795,301.410,-74.697,-177.030,8.733,148.870
C06247=1136.800,301.162,-74.666,-177.033,8.729,148.870
C06248=1136.804,300.914,-74.635,-177.035,8.726,148.870
C06249=1136.808,300.666,-74.603,-177.038,8.722,148.869
C06250=1136.812,300.418,-74.572,-177.041,8.719,148.869
C06251=1136.816,300.170,-74.541,-177.043,8.716,148.869
C06252=1136.821,299.922,-74.510,-177.046,8.712,148.869
C06253=1136.825,299.674,-74.479,-177.049,8.708,148.869
C06254=1136.829,299.426,-74.447,-177.052,8.705,148.869
C06255=1136.833,299.178,-74.416,-177.054,8.701,148.869
C06256=1136.838,298.930,-74.385,-177.057,8.698,148.869
C06257=1136.841,298.682,-74.354,-177.060,8.694,148.869
C06258=1136.845,298.434,-74.323,-177.062,8.691,148.868
C06259=1136.849,298.185,-74.292,-177.065,8.687,148.868
C06260=1136.854,297.938,-74.261,-177.068,8.684,148.868
C06261=1136.858,297.690,-74.230,-177.070,8.681,148.868
C06262=1136.862,297.441,-74.199,-177.073,8.677,148.868
C06263=1136.867,297.193,-74.168,-177.076,8.674,148.868
C06264=1136.871,296.945,-74.136,-177.079,8.670,148.868
C06265=1136.875,296.698,-74.106,-177.081,8.667,148.867
C06266=1136.879,296.450,-74.075,-177.084,8.663,148.867
C06267=1136.883,296.201,-74.044,-177.087,8.660,148.867
C06268=1136.888,295.953,-74.013,-177.090,8.656,148.867
C06269=1136.891,295.706,-73.983,-177.092,8.653,148.867
C06270=1136.895,295.457,-73.951,-177.095,8.649,148.867
C06271=1136.900,295.209,-73.921,-177.098,8.646,148.867
C06272=1136.904,294.961,-73.889,-177.101,8.642,148.867
C06273=1136.908,294.713,-73.859,-177.103,8.639,148.867
C06274=1136.912,294.465,-73.829,-177.106,8.636,148.866
C06275=1136.916,294.217,-73.797,-177.109,8.632,148.866
C06276=1136.921,293.969,-73.767,-177.111,8.629,148.866
C06277=1136.925,293.721,-73.736,-177.114,8.626,148.866
C06278=1136.929,293.472,-73.705,-177.117,8.622,148.866
C06279=1136.934,293.224,-73.675,-177.119,8.619,148.866
C06280=1136.937,292.977,-73.644,-177.122,8.615,148.866
C06281=1136.941,292.728,-73.613,-177.125,8.612,148.866
C06282=1136.946,292.480,-73.583,-177.128,8.608,148.866
C06283=1136.950,292.232,-73.552,-177.130,8.605,148.865
C06284=1136.955,291.984,-73.522,-177.133,8.601,148.865
C06285=1136.958,291.736,-73.491,-177.136,8.598,148.865
C06286=1136.962,291.488,-73.460,-177.138,8.595,148.865
C06287=1136.967,291.240,-73.430,-177.141,8.591,148.865
C06288=1136.970,290.992,-73.399,-177.144,8.588,148.865
C06289=1136.975,290.743,-73.369,-177.146,8.585,148.865
C06290=1136.979,290.496,-73.339,-177.149,8.581,148.865
C06291=1136.984,290.248,-73.308,-177.152,8.578,148.865
C06292=1136.988,289.999,-73.277,-177.154,8.575,148.865
C06293=1136.992,289.751,-73.247,-177.157,8.571,148.865
C06294=1136.996,289.503,-73.216,-177.160,8.568,148.865
C06295=1137.000,289.255,-73.187,-177.163,8.565,148.864
C06296=1137.005,289.007,-73.156,-177.166,8.561,148.864
C06297=1137.008,288.759,-73.125,-177.168,8.558,148.864
C06298=1137.013,288.511,-73.094,-177.171,8.555,148.864
C06299=1137.017,288.263,-73.065,-177.174,8.551,148.864
C06300=1137.022,288.015,-73.034,-177.176,8.547,148.864
C06301=1137.026,287.767,-73.004,-177.179,8.544,148.864
C06302=1137.031,287.491,-72.971,-177.182,8.540,148.864
C06303=1137.035,287.215,-72.937,-177.185,8.537,148.864
C06304=1137.039,286.939,-72.903,-177.188,8.532,148.864
C06305=1137.044,286.664,-72.870,-177.192,8.529,148.864
C06306=1137.048,286.416,-72.840,-177.194,8.525,148.863
C06307=1137.053,286.167,-72.809,-177.197,8.523,148.863
C06308=1137.057,285.919,-72.779,-177.199,8.519,148.863
C06309=1137.061,285.671,-72.748,-177.203,8.516,148.863
C06310=1137.065,285.423,-72.719,-177.205,8.512,148.863
C06311=1137.070,285.175,-72.688,-177.208,8.509,148.863
C06312=1137.074,284.927,-72.659,-177.211,8.505,148.863
C06313=1137.078,284.679,-72.629,-177.213,8.502,148.863
C06314=1137.083,284.431,-72.599,-177.216,8.499,148.863
C06315=1137.087,284.183,-72.568,-177.219,8.495,148.863
C06316=1137.090,283.934,-72.539,-177.222,8.492,148.863
C06317=1137.095,283.686,-72.508,-177.224,8.489,148.863
C06318=1137.099,283.438,-72.478,-177.227,8.486,148.863
C06319=1137.103,283.190,-72.449,-177.230,8.482,148.863
C06320=1137.108,282.942,-72.418,-177.232,8.479,148.862
C06321=1137.112,282.693,-72.389,-177.235,8.476,148.862
C06322=1137.116,282.446,-72.358,-177.238,8.472,148.862
C06323=1137.120,282.197,-72.329,-177.241,8.469,148.862
C06324=1137.125,281.949,-72.299,-177.243,8.466,148.862
C06325=1137.129,281.701,-72.269,-177.246,8.463,148.862
C06326=1137.133,281.453,-72.239,-177.249,8.459,148.862
C06327=1137.138,281.204,-72.209,-177.252,8.456,148.862
C06328=1137.142,280.957,-72.179,-177.255,8.453,148.862
C06329=1137.146,280.708,-72.150,-177.257,8.450,148.862
C06330=1137.150,280.460,-72.120,-177.260,8.446,148.862
C06331=1137.154,280.212,-72.091,-177.263,8.443,148.862
C06332=1137.159,279.964,-72.060,-177.265,8.440,148.862
C06333=1137.163,279.716,-72.031,-177.268,8.437,148.862
C06334=1137.167,279.467,-72.001,-177.271,8.433,148.862
C06335=1137.172,279.219,-71.972,-177.273,8.430,148.862
C06336=1137.176,278.971,-71.942,-177.276,8.427,148.862
C06337=1137.180,278.723,-71.912,-177.279,8.424,148.862
C06338=1137.185,278.475,-71.882,-177.282,8.420,148.861
C06339=1137.189,278.226,-71.853,-177.285,8.417,148.862
C06340=1137.193,277.978,-71.823,-177.287,8.413,148.861
C06341=1137.197,277.730,-71.794,-177.290,8.411,148.861
C06342=1137.201,277.482,-71.764,-177.293,8.407,148.861
C06343=1137.206,277.233,-71.735,-177.296,8.404,148.861
C06344=1137.210,276.985,-71.705,-177.298,8.401,148.861
C06345=1137.214,276.737,-71.676,-177.301,8.397,148.861
C06346=1137.218,276.488,-71.646,-177.304,8.394,148.861
C06347=1137.222,276.240,-71.617,-177.307,8.390,148.861
C06348=1137.226,275.992,-71.587,-177.309,8.387,148.861
C06349=1137.231,275.744,-71.558,-177.312,8.385,148.861
C06350=1137.235,275.495,-71.529,-177.315,8.381,148.861
C06351=1137.239,275.247,-71.499,-177.318,8.378,148.861
C06352=1137.243,274.999,-71.470,-177.320,8.374,148.861
C06353=1137.248,274.751,-71.441,-177.323,8.371,148.861
C06354=1137.252,274.503,-71.411,-177.326,8.368,148.861
C06355=1137.256,274.255,-71.382,-177.329,8.364,148.861
C06356=1137.260,274.007,-71.352,-177.331,8.362,148.861
C06357=1137.265,273.758,-71.323,-177.334,8.359,148.861
C06358=1137.269,273.510,-71.293,-177.337,8.355,148.861
C06359=1137.273,273.262,-71.264,-177.340,8.352,148.861
C06360=1137.278,273.013,-71.235,-177.343,8.349,148.861
C06361=1137.282,272.765,-71.206,-177.345,8.345,148.861
C06362=1137.286,272.517,-71.177,-177.348,8.342,148.861
C06363=1137.291,272.269,-71.147,-177.351,8.338,148.861
C06364=1137.295,272.020,-71.118,-177.354,8.336,148.861
C06365=1137.299,271.772,-71.089,-177.356,8.333,148.861
C06366=1137.304,271.523,-71.059,-177.359,8.329,148.860
C06367=1137.308,271.276,-71.031,-177.362,8.326,148.861
C06368=1137.312,271.028,-71.002,-177.365,8.323,148.861
C06369=1137.316,270.779,-70.973,-177.367,8.319,148.860
C06370=1137.320,270.531,-70.943,-177.370,8.317,148.860
C06371=1137.325,270.282,-70.914,-177.373,8.314,148.861
C06372=1137.330,270.034,-70.885,-177.375,8.310,148.860
C06373=1137.334,269.786,-70.856,-177.379,8.307,148.860
C06374=1137.337,269.538,-70.827,-177.381,8.304,148.860
C06375=1137.342,269.289,-70.798,-177.384,8.300,148.860
C06376=1137.346,269.041,-70.769,-177.387,8.298,148.860
C06377=1137.351,268.793,-70.740,-177.389,8.295,148.860
C06378=1137.355,268.544,-70.711,-177.392,8.292,148.860
C06379=1137.359,268.296,-70.682,-177.395,8.288,148.860
C06380=1137.363,268.047,-70.654,-177.398,8.285,148.860
C06381=1137.368,267.800,-70.624,-177.401,8.282,148.860
C06382=1137.372,267.551,-70.596,-177.403,8.279,148.860
C06383=1137.376,267.303,-70.567,-177.406,8.276,148.860
C06384=1137.381,267.055,-70.539,-177.409,8.272,148.860
C06385=1137.385,266.807,-70.509,-177.412,8.269,148.860
C06386=1137.389,266.558,-70.481,-177.414,8.266,148.860
C06387=1137.393,266.310,-70.451,-177.417,8.263,148.860
C06388=1137.398,266.062,-70.423,-177.420,8.260,148.860
C06389=1137.402,265.813,-70.394,-177.422,8.257,148.860
C06390=1137.406,265.565,-70.366,-177.426,8.253,148.860
C06391=1137.411,265.317,-70.337,-177.428,8.250,148.860
C06392=1137.415,265.068,-70.308,-177.431,8.247,148.860
C06393=1137.419,264.820,-70.280,-177.434,8.244,148.860
C06394=1137.424,264.572,-70.250,-177.436,8.241,148.860
C06395=1137.428,264.324,-70.222,-177.439,8.238,148.860
C06396=1137.432,264.075,-70.194,-177.442,8.234,148.860
C06397=1137.437,263.827,-70.164,-177.445,8.231,148.860
C06398=1137.441,263.579,-70.136,-177.448,8.228,148.860
C06399=1137.445,263.330,-70.108,-177.450,8.225,148.860
C06400=1137.450,263.082,-70.080,-177.453,8.222,148.860
C06401=1137.454,262.834,-70.050,-177.456,8.219,148.860
C06402=1137.459,262.585,-70.022,-177.458,8.216,148.860
C06403=1137.463,262.337,-69.994,-177.462,8.212,148.860
C06404=1137.467,262.088,-69.965,-177.465,8.209,148.860
C06405=1137.471,261.841,-69.937,-177.467,8.206,148.860
C06406=1137.476,261.566,-69.905,-177.470,8.203,148.860
C06407=1137.481,261.293,-69.874,-177.473,8.199,148.860
C06408=1137.486,261.019,-69.843,-177.476,8.196,148.860
C06409=1137.490,260.746,-69.811,-177.479,8.193,148.860
C06410=1137.495,260.498,-69.783,-177.482,8.190,148.860
C06411=1137.499,260.249,-69.755,-177.484,8.187,148.860
C06412=1137.504,260.001,-69.726,-177.487,8.184,148.860
C06413=1137.507,259.752,-69.698,-177.491,8.180,148.860
C06414=1137.512,259.503,-69.670,-177.493,8.177,148.861
C06415=1137.516,259.256,-69.642,-177.496,8.174,148.860
C06416=1137.520,259.007,-69.614,-177.499,8.171,148.860
C06417=1137.525,258.759,-69.585,-177.501,8.168,148.861
C06418=1137.529,258.510,-69.557,-177.504,8.165,148.861
C06419=1137.534,258.262,-69.529,-177.507,8.162,148.861
C06420=1137.538,258.013,-69.501,-177.509,8.159,148.861
C06421=1137.542,257.766,-69.473,-177.513,8.155,148.861
C06422=1137.546,257.517,-69.444,-177.515,8.152,148.861
C06423=1137.551,257.269,-69.416,-177.518,8.149,148.861
C06424=1137.555,257.020,-69.388,-177.521,8.146,148.861
C06425=1137.560,256.772,-69.360,-177.524,8.144,148.861
C06426=1137.563,256.523,-69.332,-177.526,8.140,148.861
C06427=1137.569,256.275,-69.303,-177.529,8.137,148.861
C06428=1137.572,256.027,-69.275,-177.532,8.134,148.861
C06429=1137.577,255.779,-69.247,-177.535,8.132,148.861
C06430=1137.581,255.529,-69.219,-177.537,8.129,148.861
C06431=1137.586,255.281,-69.192,-177.541,8.125,148.861
C06432=1137.590,255.033,-69.163,-177.543,8.122,148.861
C06433=1137.594,254.785,-69.136,-177.546,8.119,148.861
C06434=1137.599,254.537,-69.107,-177.549,8.116,148.861
C06435=1137.603,254.288,-69.080,-177.551,8.113,148.861
C06436=1137.607,254.040,-69.052,-177.554,8.110,148.861
C06437=1137.611,253.791,-69.024,-177.557,8.107,148.861
C06438=1137.616,253.543,-68.996,-177.559,8.104,148.861
C06439=1137.620,253.294,-68.968,-177.562,8.101,148.861
C06440=1137.625,253.046,-68.940,-177.565,8.098,148.861
C06441=1137.629,252.798,-68.913,-177.568,8.095,148.861
C06442=1137.633,252.549,-68.884,-177.571,8.091,148.861
C06443=1137.638,252.301,-68.857,-177.574,8.088,148.861
C06444=1137.642,252.052,-68.829,-177.577,8.085,148.861
C06445=1137.646,251.804,-68.801,-177.579,8.082,148.861
C06446=1137.651,251.556,-68.774,-177.582,8.079,148.861
C06447=1137.655,251.307,-68.746,-177.585,8.076,148.861
C06448=1137.660,251.058,-68.718,-177.588,8.074,148.862
C06449=1137.664,250.810,-68.690,-177.590,8.071,148.862
C06450=1137.668,250.562,-68.662,-177.593,8.068,148.862
C06451=1137.673,250.313,-68.635,-177.596,8.065,148.862
C06452=1137.677,250.065,-68.607,-177.599,8.062,148.862
C06453=1137.681,249.816,-68.580,-177.602,8.059,148.862
C06454=1137.686,249.568,-68.552,-177.604,8.056,148.862
C06455=1137.690,249.319,-68.525,-177.607,8.053,148.862
C06456=1137.694,249.071,-68.497,-177.609,8.050,148.862
C06457=1137.699,248.823,-68.470,-177.612,8.047,148.862
C06458=1137.703,248.575,-68.442,-177.616,8.043,148.862
C06459=1137.707,248.326,-68.415,-177.618,8.040,148.862
C06460=1137.712,248.078,-68.386,-177.621,8.037,148.862
C06461=1137.717,247.829,-68.359,-177.624,8.034,148.862
C06462=1137.721,247.580,-68.332,-177.627,8.032,148.862
C06463=1137.725,247.332,-68.304,-177.630,8.029,148.862
C06464=1137.730,247.084,-68.277,-177.632,8.026,148.862
C06465=1137.734,246.836,-68.249,-177.635,8.022,148.862
C06466=1137.738,246.586,-68.222,-177.638,8.020,148.862
C06467=1137.743,246.338,-68.195,-177.640,8.017,148.862
C06468=1137.747,246.090,-68.167,-177.643,8.014,148.863
C06469=1137.751,245.842,-68.140,-177.646,8.011,148.863
C06470=1137.755,245.593,-68.113,-177.649,8.008,148.863
C06471=1137.760,245.344,-68.086,-177.652,8.005,148.863
C06472=1137.764,245.096,-68.058,-177.654,8.002,148.863
C06473=1137.769,244.848,-68.031,-177.657,7.999,148.863
C06474=1137.773,244.599,-68.004,-177.660,7.996,148.863
C06475=1137.778,244.350,-67.976,-177.663,7.993,148.863
C06476=1137.782,244.102,-67.949,-177.666,7.990,148.863
C06477=1137.787,243.854,-67.922,-177.668,7.988,148.863
C06478=1137.791,243.605,-67.895,-177.671,7.985,148.863
C06479=1137.795,243.356,-67.867,-177.674,7.982,148.863
C06480=1137.799,243.108,-67.841,-177.677,7.979,148.863
C06481=1137.804,242.860,-67.813,-177.680,7.976,148.864
C06482=1137.808,242.612,-67.786,-177.682,7.973,148.863
C06483=1137.813,242.363,-67.759,-177.685,7.970,148.863
C06484=1137.817,242.114,-67.731,-177.688,7.967,148.864
C06485=1137.822,241.865,-67.704,-177.690,7.964,148.864
C06486=1137.825,241.617,-67.678,-177.693,7.961,148.864
C06487=1137.830,241.369,-67.651,-177.696,7.958,148.864
C06488=1137.835,241.120,-67.624,-177.699,7.955,148.864
C06489=1137.839,240.872,-67.597,-177.702,7.952,148.864
C06490=1137.843,240.624,-67.570,-177.704,7.949,148.864
C06491=1137.847,240.374,-67.543,-177.707,7.946,148.864
C06492=1137.852,240.126,-67.516,-177.710,7.944,148.864
C06493=1137.857,239.877,-67.489,-177.713,7.941,148.864
C06494=1137.861,239.629,-67.462,-177.716,7.938,148.864
C06495=1137.865,239.381,-67.435,-177.718,7.935,148.864
C06496=1137.870,239.132,-67.408,-177.721,7.932,148.865
C06497=1137.875,238.884,-67.381,-177.724,7.929,148.865
C06498=1137.879,238.635,-67.355,-177.727,7.926,148.865
C06499=1137.883,238.387,-67.327,-177.730,7.923,148.865
C06500=1137.887,238.138,-67.300,-177.732,7.920,148.865
C06501=1137.891,237.890,-67.274,-177.735,7.917,148.865
C06502=1137.896,237.641,-67.247,-177.738,7.914,148.865
C06503=1137.901,237.392,-67.220,-177.741,7.911,148.865
C06504=1137.905,237.144,-67.194,-177.744,7.909,148.865
C06505=1137.909,236.895,-67.167,-177.746,7.906,148.865
C06506=1137.914,236.647,-67.140,-177.749,7.903,148.865
C06507=1137.918,236.399,-67.113,-177.752,7.900,148.865
C06508=1137.923,236.149,-67.087,-177.755,7.897,148.866
C06509=1137.927,235.901,-67.060,-177.758,7.894,148.866
C06510=1137.932,235.630,-67.031,-177.760,7.891,148.866
C06511=1137.936,235.357,-67.001,-177.764,7.888,148.866
C06512=1137.942,235.085,-66.973,-177.767,7.885,148.866
C06513=1137.946,234.814,-66.944,-177.770,7.882,148.866
C06514=1137.951,234.565,-66.917,-177.773,7.879,148.866
C06515=1137.956,234.317,-66.890,-177.775,7.876,148.866
C06516=1137.960,234.068,-66.864,-177.778,7.873,148.866
C06517=1137.964,233.820,-66.837,-177.781,7.870,148.866
C06518=1137.969,233.571,-66.811,-177.784,7.867,148.867
C06519=1137.973,233.322,-66.784,-177.787,7.864,148.867
C06520=1137.977,233.074,-66.758,-177.789,7.862,148.867
C06521=1137.982,232.825,-66.731,-177.792,7.859,148.867
C06522=1137.986,232.577,-66.705,-177.795,7.856,148.867
C06523=1137.991,232.328,-66.678,-177.798,7.853,148.867
C06524=1137.995,232.080,-66.652,-177.801,7.850,148.867
C06525=1138.000,231.831,-66.625,-177.804,7.847,148.867
C06526=1138.004,231.582,-66.599,-177.807,7.844,148.867
C06527=1138.008,231.334,-66.573,-177.810,7.842,148.868
C06528=1138.013,231.085,-66.546,-177.812,7.839,148.868
C06529=1138.017,230.837,-66.520,-177.815,7.837,148.868
C06530=1138.022,230.588,-66.494,-177.817,7.834,148.868
C06531=1138.026,230.340,-66.467,-177.820,7.831,148.868
C06532=1138.031,230.091,-66.441,-177.823,7.828,148.868
C06533=1138.035,229.842,-66.415,-177.826,7.825,148.868
C06534=1138.039,229.594,-66.389,-177.829,7.822,148.868
C06535=1138.044,229.345,-66.363,-177.831,7.819,148.868
C06536=1138.048,229.097,-66.336,-177.834,7.816,148.868
C06537=1138.052,228.848,-66.310,-177.837,7.813,148.868
C06538=1138.057,228.599,-66.284,-177.840,7.811,148.869
C06539=1138.061,228.351,-66.258,-177.843,7.808,148.869
C06540=1138.066,228.103,-66.232,-177.845,7.806,148.869
C06541=1138.071,227.854,-66.205,-177.848,7.803,148.869
C06542=1138.075,227.605,-66.179,-177.851,7.800,148.869
C06543=1138.079,227.356,-66.154,-177.854,7.797,148.869
C06544=1138.084,227.107,-66.127,-177.857,7.794,148.869
C06545=1138.088,226.859,-66.101,-177.859,7.791,148.869
C06546=1138.093,226.611,-66.075,-177.862,7.788,148.869
C06547=1138.097,226.362,-66.050,-177.865,7.785,148.870
C06548=1138.102,226.113,-66.023,-177.868,7.783,148.870
C06549=1138.106,225.865,-65.997,-177.871,7.780,148.870
C06550=1138.110,225.616,-65.971,-177.874,7.777,148.870
C06551=1138.115,225.368,-65.946,-177.876,7.775,148.870
C06552=1138.120,225.119,-65.919,-177.879,7.772,148.870
C06553=1138.124,224.870,-65.894,-177.882,7.769,148.870
C06554=1138.128,224.622,-65.867,-177.884,7.766,148.870
C06555=1138.132,224.373,-65.841,-177.888,7.764,148.871
C06556=1138.137,224.125,-65.816,-177.891,7.761,148.871
C06557=1138.142,223.876,-65.790,-177.893,7.758,148.871
C06558=1138.146,223.627,-65.764,-177.896,7.755,148.871
C06559=1138.151,223.378,-65.738,-177.898,7.753,148.871
C06560=1138.156,223.130,-65.713,-177.901,7.750,148.871
C06561=1138.160,222.881,-65.687,-177.904,7.747,148.871
C06562=1138.164,222.633,-65.661,-177.907,7.744,148.872
C06563=1138.168,222.384,-65.635,-177.910,7.742,148.872
C06564=1138.173,222.136,-65.609,-177.913,7.739,148.872
C06565=1138.178,221.887,-65.583,-177.916,7.736,148.872
C06566=1138.182,221.638,-65.557,-177.918,7.733,148.872
C06567=1138.187,221.390,-65.532,-177.921,7.731,148.872
C06568=1138.191,221.141,-65.507,-177.924,7.728,148.872
C06569=1138.195,220.892,-65.481,-177.927,7.725,148.873
C06570=1138.200,220.643,-65.455,-177.930,7.722,148.873
C06571=1138.205,220.395,-65.430,-177.932,7.719,148.873
C06572=1138.209,220.146,-65.404,-177.935,7.717,148.873
C06573=1138.213,219.897,-65.378,-177.938,7.714,148.873
C06574=1138.218,219.649,-65.353,-177.941,7.712,148.873
C06575=1138.222,219.401,-65.327,-177.943,7.709,148.873
C06576=1138.226,219.152,-65.302,-177.946,7.706,148.873
C06577=1138.231,218.904,-65.276,-177.949,7.703,148.874
C06578=1138.236,218.654,-65.251,-177.952,7.700,148.874
C06579=1138.240,218.405,-65.225,-177.955,7.698,148.874
C06580=1138.245,218.157,-65.200,-177.957,7.696,148.874
C06581=1138.249,217.909,-65.174,-177.960,7.693,148.874
C06582=1138.253,217.660,-65.149,-177.963,7.690,148.874
C06583=1138.258,217.412,-65.123,-177.966,7.687,148.874
C06584=1138.262,217.162,-65.098,-177.969,7.684,148.875
C06585=1138.267,216.914,-65.073,-177.972,7.681,148.875
C06586=1138.272,216.665,-65.047,-177.974,7.679,148.875
C06587=1138.276,216.416,-65.022,-177.977,7.676,148.875
C06588=1138.281,216.168,-64.997,-177.980,7.674,148.875
C06589=1138.284,215.919,-64.971,-177.983,7.671,148.875
C06590=1138.289,215.671,-64.946,-177.986,7.668,148.876
C06591=1138.294,215.422,-64.921,-177.989,7.665,148.876
C06592=1138.298,215.173,-64.895,-177.991,7.663,148.876
C06593=1138.303,214.925,-64.870,-177.994,7.661,148.876
C06594=1138.307,214.675,-64.845,-177.997,7.658,148.876
C06595=1138.312,214.427,-64.819,-178.000,7.655,148.876
C06596=1138.317,214.178,-64.794,-178.003,7.652,148.876
C06597=1138.321,213.930,-64.770,-178.005,7.650,148.877
C06598=1138.325,213.681,-64.744,-178.008,7.647,148.877
C06599=1138.330,213.433,-64.719,-178.011,7.644,148.877
C06600=1138.334,213.184,-64.693,-178.014,7.641,148.877
C06601=1138.339,212.934,-64.668,-178.017,7.639,148.877
C06602=1138.343,212.687,-64.644,-178.019,7.637,148.877
C06603=1138.347,212.437,-64.619,-178.022,7.634,148.878
C06604=1138.352,212.189,-64.593,-178.025,7.631,148.878
C06605=1138.357,211.940,-64.568,-178.028,7.628,148.878
C06606=1138.361,211.692,-64.543,-178.031,7.625,148.878
C06607=1138.365,211.442,-64.518,-178.033,7.623,148.878
C06608=1138.370,211.194,-64.493,-178.036,7.620,148.878
C06609=1138.375,210.945,-64.468,-178.039,7.618,148.879
C06610=1138.379,210.696,-64.444,-178.042,7.615,148.879
C06611=1138.384,210.448,-64.418,-178.044,7.613,148.879
C06612=1138.389,210.199,-64.393,-178.047,7.610,148.879
C06613=1138.393,209.951,-64.369,-178.050,7.607,148.879
C06614=1138.398,209.680,-64.341,-178.053,7.605,148.879
C06615=1138.402,209.409,-64.314,-178.056,7.602,148.880
C06616=1138.408,209.139,-64.287,-178.059,7.599,148.880
C06617=1138.412,208.868,-64.260,-178.062,7.597,148.880
C06618=1138.417,208.619,-64.235,-178.065,7.594,148.880
C06619=1138.421,208.370,-64.211,-178.068,7.591,148.880
C06620=1138.426,208.122,-64.186,-178.071,7.588,148.880
C06621=1138.431,207.873,-64.161,-178.074,7.586,148.881
C06622=1138.435,207.624,-64.136,-178.076,7.583,148.881
C06623=1138.440,207.376,-64.112,-178.079,7.580,148.881
C06624=1138.444,207.127,-64.086,-178.082,7.578,148.881
C06625=1138.449,206.878,-64.062,-178.085,7.576,148.881
C06626=1138.454,206.630,-64.037,-178.087,7.573,148.882
C06627=1138.458,206.380,-64.013,-178.091,7.570,148.882
C06628=1138.463,206.132,-63.988,-178.094,7.567,148.882
C06629=1138.466,205.883,-63.963,-178.096,7.565,148.882
C06630=1138.471,205.635,-63.938,-178.099,7.563,148.882
C06631=1138.476,205.386,-63.914,-178.102,7.560,148.883
C06632=1138.480,205.137,-63.889,-178.105,7.557,148.883
C06633=1138.485,204.888,-63.865,-178.107,7.555,148.883
C06634=1138.490,204.640,-63.841,-178.110,7.552,148.883
C06635=1138.494,204.390,-63.815,-178.113,7.549,148.883
C06636=1138.499,204.142,-63.791,-178.116,7.547,148.884
C06637=1138.504,203.893,-63.767,-178.118,7.545,148.884
C06638=1138.507,203.644,-63.742,-178.121,7.542,148.884
C06639=1138.512,203.396,-63.717,-178.125,7.539,148.884
C06640=1138.517,203.147,-63.693,-178.127,7.537,148.884
C06641=1138.521,202.898,-63.668,-178.130,7.534,148.884
C06642=1138.526,202.650,-63.644,-178.133,7.532,148.885
C06643=1138.530,202.401,-63.620,-178.136,7.529,148.885
C06644=1138.535,202.152,-63.595,-178.138,7.527,148.885
C06645=1138.539,201.903,-63.571,-178.141,7.524,148.885
C06646=1138.544,201.654,-63.547,-178.144,7.521,148.885
C06647=1138.549,201.406,-63.523,-178.147,7.520,148.886
C06648=1138.553,201.156,-63.498,-178.150,7.517,148.886
C06649=1138.558,200.908,-63.473,-178.152,7.514,148.886
C06650=1138.562,200.659,-63.449,-178.155,7.512,148.886
C06651=1138.567,200.411,-63.425,-178.158,7.509,148.886
C06652=1138.571,200.161,-63.400,-178.161,7.507,148.887
C06653=1138.576,199.913,-63.376,-178.164,7.504,148.887
C06654=1138.580,199.665,-63.352,-178.166,7.502,148.887
C06655=1138.585,199.415,-63.328,-178.169,7.499,148.887
C06656=1138.589,199.166,-63.304,-178.172,7.496,148.887
C06657=1138.594,198.918,-63.280,-178.175,7.494,148.888
C06658=1138.599,198.669,-63.255,-178.178,7.491,148.888
C06659=1138.603,198.421,-63.231,-178.181,7.489,148.888
C06660=1138.608,198.172,-63.208,-178.183,7.487,148.888
C06661=1138.612,197.922,-63.183,-178.186,7.484,148.888
C06662=1138.617,197.674,-63.158,-178.189,7.481,148.889
C06663=1138.621,197.425,-63.134,-178.192,7.479,148.889
C06664=1138.626,197.176,-63.111,-178.195,7.477,148.889
C06665=1138.630,196.928,-63.087,-178.198,7.474,148.889
C06666=1138.635,196.678,-63.062,-178.200,7.472,148.889
C06667=1138.639,196.429,-63.038,-178.203,7.469,148.890
C06668=1138.644,196.181,-63.014,-178.206,7.466,148.890
C06669=1138.648,195.933,-62.990,-178.209,7.465,148.890
C06670=1138.654,195.683,-62.966,-178.211,7.462,148.890
C06671=1138.658,195.435,-62.942,-178.215,7.459,148.891
C06672=1138.662,195.186,-62.918,-178.217,7.457,148.891
C06673=1138.667,194.937,-62.895,-178.220,7.454,148.891
C06674=1138.671,194.688,-62.870,-178.223,7.452,148.891
C06675=1138.676,194.439,-62.847,-178.225,7.450,148.891
C06676=1138.681,194.191,-62.822,-178.229,7.447,148.892
C06677=1138.685,193.941,-62.799,-178.231,7.444,148.892
C06678=1138.690,193.693,-62.775,-178.234,7.442,148.892
C06679=1138.694,193.445,-62.751,-178.237,7.439,148.892
C06680=1138.699,193.196,-62.728,-178.240,7.438,148.893
C06681=1138.703,192.947,-62.703,-178.242,7.435,148.893
C06682=1138.707,192.697,-62.680,-178.246,7.432,148.893
C06683=1138.712,192.448,-62.656,-178.248,7.430,148.893
C06684=1138.717,192.200,-62.632,-178.251,7.427,148.893
C06685=1138.722,191.951,-62.608,-178.254,7.425,148.894
C06686=1138.726,191.702,-62.584,-178.256,7.423,148.894
C06687=1138.731,191.453,-62.561,-178.260,7.420,148.894
C06688=1138.735,191.205,-62.537,-178.262,7.417,148.894
C06689=1138.740,190.956,-62.513,-178.265,7.416,148.895
C06690=1138.745,190.707,-62.490,-178.268,7.413,148.895
C06691=1138.749,190.458,-62.466,-178.271,7.411,148.895
C06692=1138.754,190.209,-62.443,-178.273,7.408,148.895
C06693=1138.758,189.961,-62.419,-178.277,7.405,148.896
C06694=1138.763,189.712,-62.395,-178.279,7.403,148.896
C06695=1138.768,189.463,-62.372,-178.282,7.401,148.896
C06696=1138.772,189.214,-62.349,-178.284,7.399,148.896
C06697=1138.777,188.965,-62.324,-178.288,7.396,148.897
C06698=1138.782,188.716,-62.301,-178.291,7.393,148.897
C06699=1138.786,188.467,-62.278,-178.293,7.392,148.897
C06700=1138.791,188.219,-62.254,-178.296,7.389,148.897
C06701=1138.795,187.970,-62.230,-178.299,7.387,148.898
C06702=1138.800,187.721,-62.207,-178.302,7.384,148.898
C06703=1138.805,187.472,-62.184,-178.305,7.382,148.898
C06704=1138.809,187.223,-62.160,-178.307,7.379,148.898
C06705=1138.813,186.975,-62.137,-178.310,7.377,148.898
C06706=1138.818,186.726,-62.113,-178.313,7.375,148.899
C06707=1138.822,186.477,-62.090,-178.316,7.372,148.899
C06708=1138.827,186.228,-62.067,-178.319,7.369,148.899
C06709=1138.832,185.979,-62.043,-178.321,7.368,148.899
C06710=1138.837,185.730,-62.020,-178.325,7.365,148.900
C06711=1138.841,185.481,-61.996,-178.327,7.363,148.900
C06712=1138.846,185.232,-61.973,-178.330,7.361,148.900
C06713=1138.850,184.983,-61.950,-178.332,7.358,148.900
C06714=1138.854,184.734,-61.926,-178.336,7.356,148.901
C06715=1138.860,184.486,-61.903,-178.338,7.353,148.901
C06716=1138.864,184.237,-61.880,-178.341,7.351,148.901
C06717=1138.869,183.988,-61.857,-178.344,7.348,148.901
C06718=1138.874,183.718,-61.832,-178.347,7.346,148.902
C06719=1138.878,183.449,-61.806,-178.350,7.344,148.902
C06720=1138.883,183.179,-61.781,-178.353,7.341,148.902
C06721=1138.889,182.909,-61.756,-178.356,7.339,148.903
C06722=1138.893,182.660,-61.733,-178.359,7.336,148.903
C06723=1138.897,182.411,-61.710,-178.362,7.334,148.903
C06724=1138.903,182.163,-61.687,-178.365,7.332,148.903
C06725=1138.907,181.914,-61.664,-178.367,7.329,148.903
C06726=1138.911,181.665,-61.641,-178.370,7.327,148.904
C06727=1138.916,181.416,-61.617,-178.373,7.325,148.904
C06728=1138.921,181.167,-61.594,-178.376,7.322,148.904
C06729=1138.926,180.918,-61.571,-178.379,7.321,148.905
C06730=1138.930,180.669,-61.549,-178.381,7.318,148.905
C06731=1138.935,180.420,-61.526,-178.385,7.315,148.905
C06732=1138.940,180.171,-61.502,-178.387,7.313,148.905
C06733=1138.944,179.923,-61.480,-178.390,7.311,148.906
C06734=1138.948,179.674,-61.456,-178.393,7.309,148.906
C06735=1138.953,179.425,-61.433,-178.396,7.306,148.906
C06736=1138.958,179.176,-61.411,-178.398,7.304,148.906
C06737=1138.963,178.927,-61.388,-178.401,7.301,148.907
C06738=1138.967,178.678,-61.365,-178.404,7.300,148.907
C06739=1138.971,178.429,-61.342,-178.407,7.297,148.907
C06740=1138.976,178.180,-61.319,-178.410,7.295,148.907
C06741=1138.981,177.932,-61.297,-178.413,7.292,148.908
C06742=1138.986,177.683,-61.273,-178.415,7.290,148.908
C06743=1138.989,177.434,-61.251,-178.418,7.288,148.908
C06744=1138.994,177.184,-61.228,-178.421,7.286,148.909
C06745=1139.000,176.936,-61.205,-178.424,7.283,148.909
C06746=1139.004,176.687,-61.182,-178.427,7.281,148.909
C06747=1139.009,176.437,-61.160,-178.429,7.279,148.909
C06748=1139.013,176.189,-61.137,-178.432,7.277,148.910
C06749=1139.018,175.940,-61.114,-178.435,7.274,148.910
C06750=1139.022,175.691,-61.092,-178.438,7.272,148.910
C06751=1139.027,175.442,-61.068,-178.441,7.270,148.911
C06752=1139.031,175.193,-61.046,-178.443,7.268,148.911
C06753=1139.037,174.944,-61.023,-178.446,7.265,148.911
C06754=1139.041,174.696,-61.001,-178.449,7.263,148.911
C06755=1139.046,174.446,-60.978,-178.452,7.261,148.912
C06756=1139.050,174.198,-60.956,-178.455,7.259,148.912
C06757=1139.055,173.948,-60.933,-178.458,7.256,148.912
C06758=1139.059,173.700,-60.910,-178.460,7.254,148.912
C06759=1139.065,173.451,-60.888,-178.463,7.252,148.913
C06760=1139.069,173.202,-60.865,-178.466,7.250,148.913
C06761=1139.074,172.952,-60.842,-178.469,7.247,148.913
C06762=1139.078,172.704,-60.820,-178.472,7.245,148.914
C06763=1139.082,172.455,-60.798,-178.475,7.243,148.914
C06764=1139.087,172.206,-60.775,-178.477,7.241,148.914
C06765=1139.092,171.957,-60.753,-178.480,7.239,148.914
C06766=1139.097,171.708,-60.730,-178.483,7.236,148.915
C06767=1139.101,171.459,-60.708,-178.485,7.234,148.915
C06768=1139.106,171.210,-60.686,-178.489,7.232,148.915
C06769=1139.111,170.961,-60.662,-178.491,7.230,148.915
C06770=1139.115,170.712,-60.640,-178.494,7.227,148.916
C06771=1139.119,170.464,-60.618,-178.497,7.226,148.916
C06772=1139.124,170.214,-60.595,-178.500,7.223,148.916
C06773=1139.129,169.966,-60.574,-178.502,7.221,148.917
C06774=1139.134,169.717,-60.550,-178.506,7.218,148.917
C06775=1139.138,169.467,-60.528,-178.508,7.217,148.917
C06776=1139.143,169.219,-60.507,-178.511,7.215,148.918
C06777=1139.147,168.970,-60.484,-178.514,7.212,148.918
C06778=1139.153,168.721,-60.462,-178.517,7.210,148.918
C06779=1139.157,168.472,-60.440,-178.520,7.207,148.918
C06780=1139.162,168.223,-60.418,-178.522,7.206,148.919
C06781=1139.167,167.974,-60.394,-178.526,7.203,148.919
C06782=1139.171,167.724,-60.372,-178.528,7.201,148.919
C06783=1139.176,167.476,-60.351,-178.531,7.199,148.920
C06784=1139.180,167.227,-60.329,-178.534,7.197,148.920
C06785=1139.186,166.978,-60.306,-178.536,7.195,148.920
C06786=1139.189,166.729,-60.284,-178.539,7.192,148.921
C06787=1139.194,166.480,-60.262,-178.542,7.191,148.921
C06788=1139.199,166.231,-60.240,-178.545,7.188,148.921
C06789=1139.204,165.982,-60.218,-178.548,7.186,148.921
C06790=1139.209,165.733,-60.196,-178.550,7.184,148.922
C06791=1139.213,165.484,-60.174,-178.554,7.182,148.922
C06792=1139.218,165.235,-60.152,-178.556,7.180,148.922
C06793=1139.222,164.987,-60.129,-178.559,7.177,148.923
C06794=1139.226,164.737,-60.107,-178.562,7.175,148.923
C06795=1139.232,164.488,-60.085,-178.565,7.173,148.923
C06796=1139.236,164.239,-60.063,-178.567,7.171,148.924
C06797=1139.241,163.990,-60.041,-178.570,7.169,148.924
C06798=1139.245,163.741,-60.019,-178.573,7.167,148.924
C06799=1139.250,163.492,-59.998,-178.576,7.164,148.924
C06800=1139.255,163.243,-59.976,-178.579,7.162,148.925
C06801=1139.259,162.994,-59.954,-178.582,7.160,148.925
C06802=1139.264,162.745,-59.932,-178.584,7.159,148.926
C06803=1139.269,162.496,-59.910,-178.587,7.156,148.926
C06804=1139.274,162.247,-59.888,-178.590,7.154,148.926
C06805=1139.279,161.998,-59.866,-178.592,7.152,148.926
C06806=1139.283,161.749,-59.844,-178.596,7.150,148.927
C06807=1139.288,161.500,-59.822,-178.598,7.148,148.927
C06808=1139.293,161.251,-59.800,-178.601,7.145,148.927
C06809=1139.297,161.002,-59.778,-178.604,7.143,148.928
C06810=1139.302,160.753,-59.757,-178.607,7.142,148.928
C06811=1139.306,160.503,-59.735,-178.610,7.139,148.928
C06812=1139.311,160.255,-59.714,-178.612,7.137,148.929
C06813=1139.316,160.006,-59.692,-178.615,7.135,148.929
C06814=1139.320,159.757,-59.670,-178.618,7.133,148.929
C06815=1139.325,159.508,-59.648,-178.621,7.131,148.929
C06816=1139.330,159.260,-59.627,-178.624,7.128,148.930
C06817=1139.335,159.010,-59.605,-178.627,7.127,148.930
C06818=1139.339,158.761,-59.584,-178.629,7.125,148.931
C06819=1139.344,158.512,-59.562,-178.632,7.122,148.931
C06820=1139.349,158.263,-59.540,-178.635,7.120,148.931
C06821=1139.353,158.014,-59.518,-178.637,7.118,148.932
C06822=1139.358,157.745,-59.495,-178.641,7.116,148.932
C06823=1139.364,157.476,-59.472,-178.644,7.113,148.932
C06824=1139.368,157.208,-59.449,-178.647,7.112,148.933
C06825=1139.374,156.938,-59.425,-178.650,7.109,148.933
C06826=1139.378,156.690,-59.404,-178.652,7.107,148.933
C06827=1139.383,156.440,-59.382,-178.656,7.105,148.933
C06828=1139.388,156.191,-59.361,-178.658,7.103,148.934
C06829=1139.393,155.942,-59.339,-178.661,7.101,148.934
C06830=1139.397,155.693,-59.318,-178.664,7.099,148.935
C06831=1139.401,155.444,-59.296,-178.667,7.097,148.935
C06832=1139.407,155.195,-59.275,-178.669,7.095,148.935
C06833=1139.411,154.945,-59.253,-178.673,7.092,148.936
C06834=1139.416,154.697,-59.232,-178.675,7.091,148.936
C06835=1139.421,154.448,-59.211,-178.678,7.089,148.936
C06836=1139.425,154.199,-59.190,-178.681,7.086,148.936
C06837=1139.430,153.949,-59.168,-178.684,7.084,148.937
C06838=1139.435,153.701,-59.147,-178.686,7.083,148.937
C06839=1139.439,153.452,-59.125,-178.689,7.081,148.938
C06840=1139.445,153.203,-59.104,-178.692,7.078,148.938
C06841=1139.448,152.954,-59.083,-178.695,7.076,148.938
C06842=1139.453,152.704,-59.062,-178.697,7.075,148.938
C06843=1139.458,152.456,-59.040,-178.701,7.072,148.939
C06844=1139.463,152.206,-59.019,-178.703,7.070,148.939
C06845=1139.468,151.957,-58.997,-178.706,7.069,148.940
C06846=1139.472,151.708,-58.977,-178.709,7.066,148.940
C06847=1139.477,151.459,-58.956,-178.711,7.064,148.940
C06848=1139.482,151.210,-58.934,-178.714,7.062,148.941
C06849=1139.487,150.960,-58.913,-178.717,7.060,148.941
C06850=1139.491,150.712,-58.891,-178.720,7.058,148.941
C06851=1139.496,150.463,-58.871,-178.723,7.056,148.942
C06852=1139.501,150.213,-58.850,-178.725,7.054,148.942
C06853=1139.505,149.965,-58.828,-178.728,7.052,148.942
C06854=1139.510,149.716,-58.807,-178.731,7.050,148.943
C06855=1139.515,149.467,-58.785,-178.734,7.048,148.943
C06856=1139.519,149.218,-58.765,-178.737,7.046,148.943
C06857=1139.524,148.968,-58.744,-178.740,7.044,148.944
C06858=1139.529,148.720,-58.722,-178.742,7.042,148.944
C06859=1139.534,148.471,-58.702,-178.745,7.040,148.944
C06860=1139.539,148.222,-58.681,-178.748,7.038,148.945
C06861=1139.543,147.972,-58.660,-178.751,7.036,148.945
C06862=1139.547,147.723,-58.639,-178.754,7.035,148.945
C06863=1139.553,147.474,-58.618,-178.757,7.032,148.946
C06864=1139.557,147.225,-58.597,-178.760,7.030,148.946
C06865=1139.562,146.976,-58.576,-178.762,7.028,148.946
C06866=1139.567,146.727,-58.555,-178.765,7.027,148.947
C06867=1139.572,146.478,-58.534,-178.768,7.024,148.947
C06868=1139.577,146.229,-58.513,-178.771,7.022,148.947
C06869=1139.581,145.979,-58.493,-178.773,7.021,148.948
C06870=1139.586,145.730,-58.472,-178.776,7.019,148.948
C06871=1139.590,145.482,-58.451,-178.779,7.016,148.949
C06872=1139.595,145.232,-58.430,-178.782,7.014,148.949
C06873=1139.600,144.983,-58.409,-178.784,7.013,148.949
C06874=1139.605,144.734,-58.388,-178.787,7.011,148.950
C06875=1139.610,144.485,-58.367,-178.790,7.008,148.950
C06876=1139.614,144.236,-58.347,-178.793,7.007,148.950
C06877=1139.619,143.987,-58.326,-178.796,7.005,148.951
C06878=1139.624,143.738,-58.306,-178.798,7.003,148.951
C06879=1139.629,143.489,-58.284,-178.802,7.001,148.951
C06880=1139.633,143.240,-58.264,-178.804,6.999,148.952
C06881=1139.637,142.991,-58.243,-178.807,6.997,148.952
C06882=1139.642,142.741,-58.222,-178.809,6.995,148.952
C06883=1139.647,142.492,-58.201,-178.813,6.993,148.953
C06884=1139.652,142.243,-58.180,-178.815,6.991,148.953
C06885=1139.656,141.994,-58.160,-178.818,6.989,148.954
C06886=1139.661,141.745,-58.139,-178.821,6.988,148.954
C06887=1139.666,141.496,-58.119,-178.824,6.986,148.954
C06888=1139.670,141.247,-58.098,-178.827,6.983,148.955
C06889=1139.675,140.998,-58.077,-178.830,6.982,148.955
C06890=1139.680,140.749,-58.057,-178.832,6.980,148.955
C06891=1139.685,140.499,-58.037,-178.835,6.978,148.956
C06892=1139.690,140.250,-58.016,-178.837,6.976,148.956
C06893=1139.694,140.001,-57.996,-178.841,6.974,148.956
C06894=1139.699,139.752,-57.975,-178.843,6.972,148.957
C06895=1139.704,139.503,-57.955,-178.846,6.970,148.957
C06896=1139.708,139.254,-57.934,-178.849,6.969,148.958
C06897=1139.714,139.005,-57.913,-178.852,6.966,148.958
C06898=1139.718,138.756,-57.893,-178.855,6.964,148.958
C06899=1139.722,138.507,-57.873,-178.858,6.963,148.959
C06900=1139.728,138.257,-57.853,-178.860,6.961,148.959
C06901=1139.733,138.009,-57.832,-178.862,6.959,148.959
C06902=1139.737,137.760,-57.812,-178.866,6.956,148.960
C06903=1139.743,137.510,-57.791,-178.868,6.955,148.960
C06904=1139.747,137.261,-57.771,-178.871,6.953,148.960
C06905=1139.752,137.012,-57.751,-178.874,6.951,148.961
C06906=1139.756,136.763,-57.731,-178.877,6.950,148.961
C06907=1139.761,136.514,-57.710,-178.879,6.948,148.962
C06908=1139.766,136.265,-57.689,-178.883,6.945,148.962
C06909=1139.770,136.015,-57.670,-178.885,6.944,148.962
C06910=1139.775,135.766,-57.649,-178.888,6.942,148.963
C06911=1139.780,135.517,-57.628,-178.891,6.940,148.963
C06912=1139.785,135.267,-57.609,-178.894,6.939,148.964
C06913=1139.790,135.019,-57.589,-178.897,6.936,148.964
C06914=1139.794,134.770,-57.568,-178.900,6.934,148.964
C06915=1139.800,134.520,-57.548,-178.902,6.933,148.965
C06916=1139.804,134.271,-57.528,-178.905,6.931,148.965
C06917=1139.809,134.022,-57.507,-178.907,6.929,148.965
C06918=1139.813,133.773,-57.488,-178.910,6.927,148.966
C06919=1139.818,133.524,-57.467,-178.913,6.926,148.966
C06920=1139.823,133.275,-57.448,-178.916,6.923,148.967
C06921=1139.828,133.026,-57.427,-178.919,6.921,148.967
C06922=1139.833,132.777,-57.407,-178.921,6.920,148.967
C06923=1139.838,132.527,-57.387,-178.924,6.918,148.968
C06924=1139.842,132.278,-57.367,-178.927,6.916,148.968
C06925=1139.847,132.029,-57.347,-178.930,6.915,148.969
C06926=1139.852,131.760,-57.325,-178.933,6.912,148.969
C06927=1139.857,131.492,-57.303,-178.936,6.910,148.969
C06928=1139.862,131.223,-57.282,-178.939,6.908,148.970
C06929=1139.868,130.955,-57.260,-178.942,6.907,148.970
C06930=1139.873,130.706,-57.241,-178.945,6.905,148.971
C06931=1139.877,130.456,-57.221,-178.948,6.903,148.971
C06932=1139.882,130.207,-57.201,-178.950,6.901,148.971
C06933=1139.887,129.958,-57.181,-178.953,6.899,148.972
C06934=1139.892,129.709,-57.161,-178.956,6.897,148.972
C06935=1139.896,129.460,-57.141,-178.959,6.895,148.972
C06936=1139.901,129.211,-57.121,-178.961,6.894,148.973
C06937=1139.905,128.961,-57.101,-178.964,6.892,148.973
C06938=1139.911,128.713,-57.082,-178.967,6.890,148.974
C06939=1139.915,128.464,-57.062,-178.970,6.888,148.974
C06940=1139.920,128.214,-57.042,-178.972,6.887,148.974
C06941=1139.925,127.964,-57.022,-178.975,6.885,148.975
C06942=1139.930,127.716,-57.002,-178.978,6.883,148.975
C06943=1139.935,127.467,-56.983,-178.981,6.881,148.976
C06944=1139.939,127.217,-56.963,-178.984,6.879,148.976
C06945=1139.944,126.968,-56.943,-178.986,6.877,148.976
C06946=1139.949,126.719,-56.923,-178.989,6.876,148.977
C06947=1139.954,126.470,-56.904,-178.992,6.874,148.977
C06948=1139.958,126.221,-56.883,-178.995,6.872,148.978
C06949=1139.964,125.972,-56.864,-178.997,6.871,148.978
C06950=1139.968,125.722,-56.844,-179.000,6.869,148.978
C06951=1139.973,125.473,-56.825,-179.003,6.867,148.979
C06952=1139.978,125.224,-56.804,-179.006,6.865,148.979
C06953=1139.983,124.975,-56.785,-179.009,6.863,148.980
C06954=1139.988,124.725,-56.765,-179.012,6.861,148.980
C06955=1139.992,124.476,-56.746,-179.014,6.860,148.980
C06956=1139.997,124.227,-56.727,-179.017,6.858,148.981
C06957=1140.001,123.978,-56.707,-179.020,6.856,148.981
C06958=1140.006,123.729,-56.687,-179.022,6.855,148.982
C06959=1140.011,123.480,-56.668,-179.025,6.853,148.982
C06960=1140.016,123.230,-56.648,-179.028,6.851,148.982
C06961=1140.021,122.981,-56.628,-179.031,6.850,148.983
C06962=1140.026,122.732,-56.610,-179.033,6.848,148.983
C06963=1140.030,122.483,-56.590,-179.037,6.846,148.984
C06964=1140.035,122.234,-56.570,-179.040,6.844,148.984
C06965=1140.040,121.985,-56.550,-179.043,6.842,148.985
C06966=1140.045,121.735,-56.531,-179.045,6.841,148.985
C06967=1140.049,121.487,-56.512,-179.048,6.839,148.985
C06968=1140.054,121.237,-56.492,-179.051,6.837,148.986
C06969=1140.059,120.987,-56.473,-179.053,6.836,148.986
C06970=1140.064,120.739,-56.453,-179.056,6.834,148.987
C06971=1140.069,120.489,-56.434,-179.059,6.832,148.987
C06972=1140.074,120.240,-56.415,-179.062,6.831,148.987
C06973=1140.078,119.991,-56.395,-179.064,6.829,148.988
C06974=1140.084,119.742,-56.376,-179.067,6.827,148.988
C06975=1140.088,119.492,-56.356,-179.070,6.825,148.989
C06976=1140.092,119.243,-56.337,-179.073,6.824,148.989
C06977=1140.098,118.994,-56.318,-179.075,6.822,148.989
C06978=1140.103,118.745,-56.298,-179.078,6.820,148.990
C06979=1140.107,118.496,-56.280,-179.081,6.819,148.990
C06980=1140.112,118.246,-56.261,-179.083,6.817,148.991
C06981=1140.118,117.997,-56.242,-179.087,6.815,148.991
C06982=1140.122,117.748,-56.222,-179.090,6.813,148.991
C06983=1140.127,117.499,-56.203,-179.092,6.811,148.992
C06984=1140.132,117.249,-56.184,-179.095,6.809,148.992
C06985=1140.136,117.000,-56.164,-179.098,6.808,148.993
C06986=1140.141,116.751,-56.145,-179.100,6.806,148.993
C06987=1140.146,116.502,-56.126,-179.104,6.805,148.994
C06988=1140.151,116.253,-56.108,-179.106,6.803,148.994
C06989=1140.155,116.003,-56.088,-179.109,6.801,148.994
C06990=1140.161,115.754,-56.069,-179.112,6.800,148.995
C06991=1140.165,115.505,-56.050,-179.115,6.798,148.995
C06992=1140.170,115.256,-56.030,-179.117,6.796,148.996
C06993=1140.175,115.007,-56.012,-179.120,6.795,148.996
C06994=1140.180,114.757,-55.993,-179.123,6.793,148.997
C06995=1140.185,114.508,-55.973,-179.125,6.791,148.997
C06996=1140.189,114.259,-55.954,-179.128,6.790,148.997
C06997=1140.195,114.010,-55.936,-179.131,6.788,148.998
C06998=1140.199,113.760,-55.917,-179.134,6.786,148.998
C06999=1140.204,113.512,-55.897,-179.136,6.785,148.999
C07000=1140.208,113.262,-55.879,-179.139,6.783,148.999
C07001=1140.214,113.013,-55.860,-179.142,6.782,149.000
C07002=1140.218,112.763,-55.840,-179.145,6.780,149.000
C07003=1140.223,112.514,-55.822,-179.148,6.778,149.000
C07004=1140.229,112.265,-55.803,-179.150,6.776,149.001
C07005=1140.233,112.016,-55.784,-179.153,6.775,149.001
C07006=1140.238,111.766,-55.765,-179.156,6.773,149.002
C07007=1140.242,111.517,-55.746,-179.159,6.771,149.002
C07008=1140.248,111.268,-55.728,-179.161,6.770,149.002
C07009=1140.253,111.019,-55.709,-179.164,6.768,149.003
C07010=1140.257,110.770,-55.689,-179.167,6.766,149.003
C07011=1140.262,110.520,-55.671,-179.170,6.765,149.004
C07012=1140.267,110.271,-55.652,-179.172,6.763,149.004
C07013=1140.272,110.022,-55.634,-179.176,6.762,149.005
C07014=1140.277,109.773,-55.615,-179.178,6.760,149.005
C07015=1140.282,109.523,-55.596,-179.181,6.758,149.006
C07016=1140.286,109.274,-55.577,-179.184,6.757,149.006
C07017=1140.291,109.024,-55.558,-179.186,6.755,149.006
C07018=1140.296,108.776,-55.540,-179.189,6.753,149.007
C07019=1140.301,108.526,-55.522,-179.192,6.752,149.007
C07020=1140.306,108.277,-55.502,-179.195,6.750,149.008
C07021=1140.310,108.028,-55.484,-179.197,6.749,149.008
C07022=1140.316,107.779,-55.465,-179.200,6.747,149.008
C07023=1140.320,107.529,-55.446,-179.203,6.746,149.009
C07024=1140.325,107.280,-55.428,-179.205,6.744,149.009
C07025=1140.330,107.031,-55.409,-179.208,6.743,149.010
C07026=1140.335,106.781,-55.391,-179.211,6.741,149.010
C07027=1140.339,106.533,-55.372,-179.214,6.739,149.011
C07028=1140.345,106.283,-55.353,-179.216,6.738,149.011
C07029=1140.349,106.034,-55.334,-179.219,6.736,149.012
C07030=1140.355,105.765,-55.314,-179.222,6.735,149.012
C07031=1140.360,105.497,-55.295,-179.225,6.733,149.013
C07032=1140.365,105.229,-55.276,-179.228,6.730,149.013
C07033=1140.370,104.961,-55.255,-179.231,6.729,149.013
C07034=1140.375,104.711,-55.236,-179.234,6.727,149.014
C07035=1140.380,104.462,-55.219,-179.237,6.726,149.014
C07036=1140.385,104.212,-55.200,-179.240,6.724,149.015
C07037=1140.389,103.963,-55.181,-179.242,6.723,149.015
C07038=1140.394,103.714,-55.163,-179.245,6.722,149.016
C07039=1140.400,103.464,-55.144,-179.247,6.720,149.016
C07040=1140.404,103.216,-55.126,-179.250,6.718,149.016
C07041=1140.409,102.966,-55.107,-179.253,6.717,149.017
C07042=1140.414,102.717,-55.089,-179.256,6.715,149.018
C07043=1140.419,102.468,-55.071,-179.259,6.714,149.018
C07044=1140.424,102.218,-55.053,-179.262,6.712,149.018
C07045=1140.429,101.969,-55.034,-179.264,6.710,149.019
C07046=1140.433,101.720,-55.016,-179.267,6.709,149.019
C07047=1140.438,101.470,-54.998,-179.270,6.707,149.020
C07048=1140.443,101.221,-54.980,-179.273,6.705,149.020
C07049=1140.449,100.972,-54.961,-179.276,6.704,149.021
C07050=1140.453,100.722,-54.943,-179.278,6.703,149.021
C07051=1140.458,100.473,-54.924,-179.281,6.701,149.022
C07052=1140.462,100.224,-54.906,-179.283,6.700,149.022
C07053=1140.467,99.975,-54.888,-179.286,6.698,149.022
C07054=1140.472,99.726,-54.870,-179.289,6.696,149.023
C07055=1140.477,99.476,-54.851,-179.292,6.695,149.023
C07056=1140.482,99.226,-54.833,-179.295,6.693,149.024
C07057=1140.487,98.977,-54.815,-179.297,6.692,149.024
C07058=1140.492,98.728,-54.797,-179.300,6.690,149.025
C07059=1140.497,98.479,-54.779,-179.302,6.689,149.025
C07060=1140.502,98.230,-54.761,-179.305,6.687,149.025
C07061=1140.506,97.980,-54.743,-179.308,6.686,149.026
C07062=1140.511,97.731,-54.725,-179.311,6.684,149.027
C07063=1140.516,97.481,-54.707,-179.314,6.683,149.027
C07064=1140.521,97.232,-54.689,-179.317,6.681,149.027
C07065=1140.526,96.983,-54.671,-179.319,6.679,149.028
C07066=1140.532,96.734,-54.653,-179.322,6.678,149.028
C07067=1140.536,96.484,-54.635,-179.325,6.676,149.029
C07068=1140.541,96.235,-54.617,-179.327,6.676,149.029
C07069=1140.546,95.985,-54.598,-179.330,6.674,149.030
C07070=1140.551,95.736,-54.580,-179.333,6.672,149.030
C07071=1140.555,95.487,-54.562,-179.336,6.671,149.031
C07072=1140.560,95.238,-54.544,-179.338,6.669,149.031
C07073=1140.565,94.989,-54.526,-179.341,6.667,149.031
C07074=1140.570,94.740,-54.508,-179.344,6.666,149.032
C07075=1140.575,94.490,-54.491,-179.346,6.665,149.032
C07076=1140.580,94.241,-54.473,-179.349,6.663,149.033
C07077=1140.585,93.991,-54.455,-179.352,6.662,149.033
C07078=1140.590,93.742,-54.437,-179.355,6.660,149.034
C07079=1140.595,93.493,-54.419,-179.357,6.658,149.034
C07080=1140.599,93.243,-54.401,-179.361,6.657,149.035
C07081=1140.604,92.994,-54.384,-179.363,6.655,149.035
C07082=1140.609,92.745,-54.366,-179.365,6.654,149.036
C07083=1140.614,92.495,-54.348,-179.368,6.653,149.036
C07084=1140.619,92.246,-54.330,-179.371,6.651,149.036
C07085=1140.624,91.997,-54.312,-179.374,6.650,149.037
C07086=1140.629,91.747,-54.295,-179.377,6.648,149.037
C07087=1140.634,91.498,-54.277,-179.380,6.646,149.038
C07088=1140.639,91.249,-54.259,-179.382,6.646,149.038
C07089=1140.643,91.000,-54.241,-179.384,6.644,149.039
C07090=1140.649,90.750,-54.224,-179.388,6.643,149.039
C07091=1140.653,90.501,-54.206,-179.390,6.641,149.040
C07092=1140.658,90.252,-54.188,-179.393,6.639,149.040
C07093=1140.663,90.002,-54.171,-179.396,6.638,149.041
C07094=1140.668,89.753,-54.153,-179.398,6.637,149.041
C07095=1140.673,89.504,-54.135,-179.401,6.635,149.042
C07096=1140.678,89.254,-54.118,-179.404,6.634,149.042
C07097=1140.682,89.005,-54.100,-179.407,6.632,149.043
C07098=1140.687,88.756,-54.083,-179.410,6.630,149.043
C07099=1140.692,88.506,-54.065,-179.412,6.630,149.043
C07100=1140.697,88.257,-54.047,-179.415,6.628,149.044
C07101=1140.702,88.007,-54.030,-179.418,6.627,149.044
C07102=1140.707,87.758,-54.013,-179.420,6.625,149.045
C07103=1140.712,87.509,-53.995,-179.423,6.623,149.045
C07104=1140.717,87.259,-53.977,-179.425,6.622,149.046
C07105=1140.722,87.010,-53.959,-179.428,6.621,149.046
C07106=1140.727,86.761,-53.942,-179.431,6.619,149.047
C07107=1140.732,86.512,-53.925,-179.434,6.618,149.047
C07108=1140.737,86.262,-53.908,-179.437,6.616,149.048
C07109=1140.742,86.013,-53.890,-179.439,6.615,149.048
C07110=1140.747,85.763,-53.873,-179.442,6.614,149.049
C07111=1140.751,85.514,-53.855,-179.445,6.612,149.049
C07112=1140.756,85.265,-53.838,-179.448,6.611,149.050
C07113=1140.761,85.016,-53.820,-179.450,6.609,149.050
C07114=1140.766,84.766,-53.803,-179.453,6.608,149.051
C07115=1140.771,84.517,-53.785,-179.456,6.607,149.051
C07116=1140.776,84.267,-53.768,-179.458,6.605,149.052
C07117=1140.781,84.019,-53.751,-179.461,6.604,149.052
C07118=1140.786,83.769,-53.734,-179.464,6.602,149.052
C07119=1140.791,83.519,-53.717,-179.466,6.601,149.053
C07120=1140.795,83.270,-53.699,-179.469,6.600,149.053
C07121=1140.801,83.021,-53.682,-179.472,6.598,149.054
C07122=1140.805,82.771,-53.664,-179.475,6.596,149.054
C07123=1140.810,82.522,-53.647,-179.477,6.596,149.055
C07124=1140.815,82.272,-53.630,-179.480,6.594,149.055
C07125=1140.821,82.024,-53.612,-179.483,6.593,149.056
C07126=1140.825,81.774,-53.596,-179.486,6.591,149.056
C07127=1140.830,81.524,-53.578,-179.488,6.590,149.057
C07128=1140.835,81.276,-53.561,-179.491,6.589,149.057
C07129=1140.840,81.026,-53.544,-179.494,6.587,149.058
C07130=1140.845,80.776,-53.526,-179.496,6.585,149.058
C07131=1140.850,80.528,-53.509,-179.499,6.585,149.059
C07132=1140.855,80.278,-53.492,-179.502,6.583,149.059
C07133=1140.859,80.029,-53.476,-179.505,6.582,149.060
C07134=1140.865,79.760,-53.457,-179.507,6.580,149.060
C07135=1140.871,79.491,-53.439,-179.511,6.579,149.061
C07136=1140.875,79.223,-53.420,-179.513,6.577,149.061
C07137=1140.881,78.955,-53.401,-179.516,6.576,149.062
C07138=1140.886,78.706,-53.385,-179.519,6.574,149.062
C07139=1140.891,78.456,-53.367,-179.521,6.573,149.063
C07140=1140.895,78.207,-53.351,-179.524,6.571,149.063
C07141=1140.901,77.957,-53.333,-179.527,6.570,149.064
C07142=1140.906,77.708,-53.317,-179.529,6.569,149.064
C07143=1140.911,77.459,-53.299,-179.532,6.568,149.065
C07144=1140.915,77.209,-53.283,-179.535,6.566,149.065
C07145=1140.920,76.960,-53.265,-179.538,6.565,149.066
C07146=1140.925,76.711,-53.249,-179.540,6.564,149.066
C07147=1140.931,76.461,-53.232,-179.543,6.562,149.067
C07148=1140.935,76.212,-53.215,-179.546,6.561,149.067
C07149=1140.940,75.962,-53.198,-179.549,6.559,149.068
C07150=1140.945,75.713,-53.181,-179.551,6.558,149.068
C07151=1140.950,75.464,-53.163,-179.554,6.557,149.069
C07152=1140.955,75.214,-53.147,-179.557,6.555,149.069
C07153=1140.960,74.966,-53.131,-179.559,6.555,149.070
C07154=1140.965,74.716,-53.113,-179.562,6.553,149.070
C07155=1140.969,74.466,-53.097,-179.565,6.551,149.070
C07156=1140.975,74.216,-53.079,-179.567,6.550,149.071
C07157=1140.980,73.968,-53.063,-179.570,6.549,149.072
C07158=1140.984,73.718,-53.046,-179.573,6.547,149.072
C07159=1140.989,73.468,-53.029,-179.576,6.546,149.072
C07160=1140.995,73.220,-53.013,-179.578,6.545,149.073
C07161=1141.000,72.970,-52.996,-179.581,6.544,149.074
C07162=1141.004,72.720,-52.979,-179.584,6.542,149.074
C07163=1141.009,72.472,-52.963,-179.586,6.541,149.074
C07164=1141.015,72.222,-52.945,-179.589,6.540,149.075
C07165=1141.019,71.972,-52.929,-179.592,6.538,149.075
C07166=1141.024,71.723,-52.913,-179.594,6.537,149.076
C07167=1141.030,71.473,-52.896,-179.597,6.536,149.076
C07168=1141.034,71.224,-52.879,-179.600,6.534,149.077
C07169=1141.039,70.975,-52.863,-179.603,6.533,149.077
C07170=1141.044,70.725,-52.846,-179.605,6.532,149.078
C07171=1141.049,70.475,-52.829,-179.608,6.530,149.078
C07172=1141.054,70.227,-52.813,-179.611,6.529,149.079
C07173=1141.058,69.977,-52.796,-179.613,6.528,149.079
C07174=1141.065,69.728,-52.780,-179.616,6.526,149.080
C07175=1141.069,69.478,-52.763,-179.619,6.525,149.080
C07176=1141.074,69.229,-52.746,-179.621,6.524,149.081
C07177=1141.079,68.979,-52.729,-179.624,6.523,149.081
C07178=1141.084,68.730,-52.713,-179.627,6.521,149.082
C07179=1141.089,68.481,-52.696,-179.629,6.521,149.082
C07180=1141.094,68.231,-52.681,-179.632,6.519,149.083
C07181=1141.098,67.982,-52.664,-179.635,6.517,149.083
C07182=1141.104,67.733,-52.647,-179.637,6.517,149.084
C07183=1141.108,67.483,-52.630,-179.640,6.515,149.084
C07184=1141.114,67.234,-52.615,-179.643,6.513,149.085
C07185=1141.118,66.984,-52.598,-179.645,6.513,149.085
C07186=1141.123,66.735,-52.581,-179.648,6.511,149.086
C07187=1141.129,66.486,-52.564,-179.651,6.510,149.086
C07188=1141.133,66.235,-52.549,-179.653,6.509,149.087
C07189=1141.139,65.987,-52.532,-179.657,6.508,149.087
C07190=1141.143,65.737,-52.516,-179.659,6.507,149.088
C07191=1141.148,65.488,-52.500,-179.661,6.505,149.088
C07192=1141.153,65.238,-52.483,-179.664,6.503,149.089
C07193=1141.159,64.989,-52.466,-179.667,6.503,149.089
C07194=1141.163,64.739,-52.450,-179.670,6.501,149.090
C07195=1141.169,64.490,-52.434,-179.672,6.500,149.090
C07196=1141.173,64.241,-52.417,-179.675,6.499,149.091
C07197=1141.178,63.991,-52.402,-179.678,6.497,149.091
C07198=1141.183,63.742,-52.385,-179.680,6.497,149.092
C07199=1141.188,63.492,-52.369,-179.683,6.495,149.092
C07200=1141.193,63.243,-52.353,-179.686,6.494,149.093
C07201=1141.198,62.993,-52.337,-179.688,6.493,149.093
C07202=1141.203,62.744,-52.321,-179.691,6.491,149.094
C07203=1141.208,62.494,-52.303,-179.694,6.490,149.094
C07204=1141.213,62.245,-52.288,-179.696,6.489,149.095
C07205=1141.218,61.996,-52.272,-179.699,6.487,149.095
C07206=1141.223,61.746,-52.256,-179.701,6.487,149.096
C07207=1141.228,61.497,-52.239,-179.704,6.485,149.096
C07208=1141.233,61.247,-52.223,-179.707,6.484,149.097
C07209=1141.238,60.998,-52.207,-179.710,6.483,149.098
C07210=1141.243,60.748,-52.191,-179.712,6.482,149.098
C07211=1141.248,60.500,-52.175,-179.715,6.481,149.098
C07212=1141.253,60.249,-52.159,-179.718,6.479,149.099
C07213=1141.258,60.001,-52.143,-179.721,6.478,149.100
C07214=1141.263,59.751,-52.127,-179.723,6.477,149.100
C07215=1141.268,59.501,-52.111,-179.725,6.475,149.100
C07216=1141.273,59.252,-52.095,-179.728,6.475,149.101
C07217=1141.278,59.002,-52.079,-179.731,6.473,149.101
C07218=1141.283,58.753,-52.062,-179.734,6.472,149.102
C07219=1141.288,58.503,-52.046,-179.736,6.471,149.103
C07220=1141.293,58.254,-52.031,-179.739,6.469,149.103
C07221=1141.298,58.004,-52.014,-179.741,6.469,149.103
C07222=1141.303,57.755,-51.999,-179.744,6.467,149.104
C07223=1141.308,57.506,-51.982,-179.747,6.466,149.105
C07224=1141.313,57.256,-51.966,-179.749,6.465,149.105
C07225=1141.317,57.007,-51.951,-179.752,6.464,149.106
C07226=1141.323,56.758,-51.935,-179.755,6.463,149.106
C07227=1141.327,56.508,-51.919,-179.757,6.461,149.107
C07228=1141.333,56.259,-51.904,-179.761,6.460,149.107
C07229=1141.338,56.009,-51.888,-179.763,6.459,149.108
C07230=1141.343,55.760,-51.871,-179.766,6.457,149.108
C07231=1141.348,55.511,-51.856,-179.768,6.457,149.109
C07232=1141.353,55.260,-51.840,-179.771,6.455,149.109
C07233=1141.358,55.012,-51.823,-179.773,6.454,149.110
C07234=1141.362,54.763,-51.808,-179.776,6.453,149.110
C07235=1141.367,54.512,-51.792,-179.778,6.452,149.111
C07236=1141.373,54.263,-51.777,-179.781,6.451,149.111
C07237=1141.378,54.014,-51.761,-179.784,6.449,149.112
C07238=1141.384,53.745,-51.744,-179.787,6.448,149.112
C07239=1141.389,53.476,-51.727,-179.790,6.447,149.113
C07240=1141.394,53.207,-51.710,-179.793,6.446,149.113
C07241=1141.400,52.939,-51.693,-179.796,6.444,149.114
C07242=1141.404,52.690,-51.678,-179.798,6.443,149.115
C07243=1141.409,52.440,-51.662,-179.801,6.442,149.115
C07244=1141.414,52.191,-51.646,-179.803,6.441,149.116
C07245=1141.420,51.942,-51.630,-179.806,6.440,149.116
C07246=1141.425,51.692,-51.614,-179.808,6.439,149.117
C07247=1141.429,51.442,-51.599,-179.812,6.438,149.117
C07248=1141.434,51.193,-51.583,-179.814,6.437,149.118
C07249=1141.440,50.944,-51.568,-179.816,6.435,149.118
C07250=1141.445,50.694,-51.552,-179.819,6.435,149.119
C07251=1141.449,50.444,-51.537,-179.822,6.433,149.119
C07252=1141.455,50.195,-51.521,-179.825,6.431,149.120
C07253=1141.460,49.946,-51.506,-179.827,6.431,149.120
C07254=1141.464,49.696,-51.489,-179.830,6.429,149.121
C07255=1141.469,49.447,-51.474,-179.832,6.428,149.121
C07256=1141.475,49.198,-51.459,-179.835,6.427,149.122
C07257=1141.480,48.948,-51.443,-179.838,6.426,149.122
C07258=1141.484,48.698,-51.428,-179.840,6.425,149.123
C07259=1141.489,48.449,-51.412,-179.843,6.424,149.123
C07260=1141.495,48.200,-51.396,-179.846,6.423,149.124
C07261=1141.499,47.951,-51.381,-179.848,6.422,149.124
C07262=1141.504,47.700,-51.365,-179.851,6.420,149.125
C07263=1141.510,47.451,-51.350,-179.853,6.420,149.125
C07264=1141.514,47.201,-51.336,-179.856,6.418,149.126
C07265=1141.520,46.952,-51.320,-179.859,6.417,149.127
C07266=1141.525,46.703,-51.304,-179.861,6.416,149.127
C07267=1141.529,46.453,-51.289,-179.864,6.415,149.127
C07268=1141.535,46.203,-51.273,-179.867,6.414,149.128
C07269=1141.539,45.954,-51.258,-179.869,6.413,149.129
C07270=1141.545,45.705,-51.243,-179.872,6.411,149.129
C07271=1141.550,45.455,-51.227,-179.874,6.411,149.130
C07272=1141.554,45.206,-51.212,-179.877,6.409,149.130
C07273=1141.560,44.956,-51.196,-179.879,6.408,149.131
C07274=1141.565,44.707,-51.182,-179.883,6.407,149.131
C07275=1141.570,44.457,-51.166,-179.885,6.406,149.132
C07276=1141.575,44.208,-51.151,-179.888,6.405,149.132
C07277=1141.580,43.959,-51.136,-179.890,6.404,149.133
C07278=1141.585,43.709,-51.120,-179.893,6.402,149.133
C07279=1141.589,43.459,-51.105,-179.896,6.402,149.134
C07280=1141.595,43.209,-51.090,-179.898,6.400,149.134
